LIN {X 0,Y 436.626,Z 302.642,A -85,B 0,C 180,E1 -16932.037,E2 -16932.037} C_VEL
LIN {X 0,Y 436.568,Z 302.656,A -85,B 0,C 180,E1 -16935.718,E2 -16935.718} C_VEL
LIN {X 0,Y 436.534,Z 302.659,A -85,B 0,C 180,E1 -16938.803,E2 -16938.803} C_VEL
LIN {X 0,Y 436.465,Z 302.663,A -85,B 0,C 180,E1 -16941.661,E2 -16941.661} C_VEL
LIN {X 0,Y 436.431,Z 302.68,A -85,B 0,C 180,E1 -16944.663,E2 -16944.663} C_VEL
LIN {X 0,Y 436.477,Z 302.669,A -85,B 0,C 180,E1 -16947.735,E2 -16947.735} C_VEL
LIN {X 0,Y 436.459,Z 302.67,A -85,B 0,C 180,E1 -16950.9,E2 -16950.9} C_VEL
LIN {X 0,Y 436.467,Z 302.658,A -85,B 0,C 180,E1 -16954.172,E2 -16954.172} C_VEL
LIN {X 0,Y 436.511,Z 302.66,A -85,B 0,C 180,E1 -16957.573,E2 -16957.573} C_VEL
LIN {X 0,Y 436.464,Z 302.674,A -85,B 0,C 180,E1 -16961.043,E2 -16961.043} C_VEL
LIN {X 0,Y 436.453,Z 302.675,A -85,B 0,C 180,E1 -16963.769,E2 -16963.769} C_VEL
LIN {X 0,Y 436.456,Z 302.678,A -85,B 0,C 180,E1 -16966.367,E2 -16966.367} C_VEL
LIN {X 0,Y 436.474,Z 302.672,A -85,B 0,C 180,E1 -16968.96,E2 -16968.96} C_VEL
LIN {X 0,Y 436.511,Z 302.67,A -85,B 0,C 180,E1 -16972.431,E2 -16972.431} C_VEL
LIN {X 0,Y 436.473,Z 302.675,A -85,B 0,C 180,E1 -16975.832,E2 -16975.832} C_VEL
LIN {X 0,Y 436.527,Z 302.878,A -85,B 0,C 180,E1 -16976.701,E2 -16976.701} C_VEL
LIN {X 0,Y 439.17,Z 313.579,A -85,B 0,C 180,E1 -16979.048,E2 -16979.048} C_VEL
LIN {X 0,Y 442.005,Z 325.849,A -85,B 0,C 180,E1 -16981.617,E2 -16981.617} C_VEL
LIN {X 0,Y 443.65,Z 334.082,A -85,B 0,C 180,E1 -16983.262,E2 -16983.262} C_VEL
LIN {X 0,Y 443.2,Z 339.732,A -85,B 0,C 180,E1 -16984.269,E2 -16984.269} C_VEL
LIN {X 0,Y 441.528,Z 353.315,A -85,B 0,C 180,E1 -16986.606,E2 -16986.606} C_VEL
LIN {X 0,Y 446.637,Z 380.69,A -85,B 0,C 180,E1 -16987.421,E2 -16987.421} C_VEL
LIN {X 0,Y 449.876,Z 402.607,A -85,B 0,C 180,E1 -16988.005,E2 -16988.005} C_VEL
LIN {X 0,Y 448.042,Z 491.581,A -85,B 0,C 180,E1 -16989.468,E2 -16989.468} C_VEL
LIN {X 0,Y 447.149,Z 506.11,A -85,B 0,C 180,E1 -16989.874,E2 -16989.874} C_VEL
LIN {X 0,Y 445.901,Z 520.039,A -85,B 0,C 180,E1 -16990.443,E2 -16990.443} C_VEL
LIN {X 0,Y 444.716,Z 532.023,A -85,B 0,C 180,E1 -16991.1,E2 -16991.1} C_VEL
LIN {X 0,Y 443.3,Z 544.152,A -85,B 0,C 180,E1 -16991.938,E2 -16991.938} C_VEL
LIN {X 0,Y 441.733,Z 555.894,A -85,B 0,C 180,E1 -16992.944,E2 -16992.944} C_VEL
LIN {X 0,Y 440.163,Z 566.666,A -85,B 0,C 180,E1 -16994.07,E2 -16994.07} C_VEL
LIN {X 0,Y 438.61,Z 577.353,A -85,B 0,C 180,E1 -16995.435,E2 -16995.435} C_VEL
LIN {X 0,Y 437.396,Z 586.21,A -85,B 0,C 180,E1 -16996.811,E2 -16996.811} C_VEL
LIN {X 0,Y 436.36,Z 594.06,A -85,B 0,C 180,E1 -16998.286,E2 -16998.286} C_VEL
LIN {X 0,Y 435.482,Z 600.731,A -85,B 0,C 180,E1 -16999.812,E2 -16999.812} C_VEL
LIN {X 0,Y 434.977,Z 605.724,A -85,B 0,C 180,E1 -17001.203,E2 -17001.203} C_VEL
LIN {X 0,Y 434.568,Z 610.914,A -85,B 0,C 180,E1 -17003.059,E2 -17003.059} C_VEL
LIN {X 0,Y 434.535,Z 612.949,A -85,B 0,C 180,E1 -17003.988,E2 -17003.988} C_VEL
LIN {X 0,Y 434.452,Z 617.176,A -85,B 0,C 180,E1 -17005.379,E2 -17005.379} C_VEL
LIN {X 0,Y 434.447,Z 621.405,A -85,B 0,C 180,E1 -17007.23,E2 -17007.23} C_VEL
LIN {X 0,Y 434.461,Z 624.028,A -85,B 0,C 180,E1 -17009.078,E2 -17009.078} C_VEL
LIN {X 0,Y 434.421,Z 625.147,A -85,B 0,C 180,E1 -17010.926,E2 -17010.926} C_VEL
LIN {X 0,Y 434.377,Z 624.813,A -85,B 0,C 180,E1 -17012.775,E2 -17012.775} C_VEL
LIN {X 0,Y 434.433,Z 623.036,A -85,B 0,C 180,E1 -17014.626,E2 -17014.626} C_VEL
LIN {X 0,Y 434.655,Z 619.805,A -85,B 0,C 180,E1 -17016.479,E2 -17016.479} C_VEL
LIN {X 0,Y 435.059,Z 615.026,A -85,B 0,C 180,E1 -17018.334,E2 -17018.334} C_VEL
LIN {X 0,Y 435.962,Z 608.502,A -85,B 0,C 180,E1 -17020.182,E2 -17020.182} C_VEL
LIN {X 0,Y 436.761,Z 602.482,A -85,B 0,C 180,E1 -17021.552,E2 -17021.552} C_VEL
LIN {X 0,Y 437.804,Z 595.077,A -85,B 0,C 180,E1 -17022.945,E2 -17022.945} C_VEL
LIN {X 0,Y 439.067,Z 586.283,A -85,B 0,C 180,E1 -17024.318,E2 -17024.318} C_VEL
LIN {X 0,Y 440.576,Z 575.698,A -85,B 0,C 180,E1 -17025.683,E2 -17025.683} C_VEL
LIN {X 0,Y 442.174,Z 563.937,A -85,B 0,C 180,E1 -17026.924,E2 -17026.924} C_VEL
LIN {X 0,Y 443.635,Z 552.309,A -85,B 0,C 180,E1 -17027.934,E2 -17027.934} C_VEL
LIN {X 0,Y 445.171,Z 539.699,A -85,B 0,C 180,E1 -17028.819,E2 -17028.819} C_VEL
LIN {X 0,Y 446.569,Z 525.705,A -85,B 0,C 180,E1 -17029.592,E2 -17029.592} C_VEL
LIN {X 0,Y 447.915,Z 510.572,A -85,B 0,C 180,E1 -17030.205,E2 -17030.205} C_VEL
LIN {X 0,Y 448.886,Z 495.971,A -85,B 0,C 180,E1 -17030.615,E2 -17030.615} C_VEL
LIN {X 0,Y 453.117,Z 405.026,A -85,B 0,C 180,E1 -17032.685,E2 -17032.685} C_VEL
LIN {X 0,Y 452.117,Z 390.827,A -85,B 0,C 180,E1 -17033.164,E2 -17033.164} C_VEL
LIN {X 0,Y 449.353,Z 368.94,A -85,B 0,C 180,E1 -17034.04,E2 -17034.04} C_VEL
LIN {X 0,Y 446.685,Z 353.618,A -85,B 0,C 180,E1 -17034.77,E2 -17034.77} C_VEL
LIN {X 0,Y 445.256,Z 335.993,A -85,B 0,C 180,E1 -17036.136,E2 -17036.136} C_VEL
LIN {X 0,Y 444.74,Z 331.395,A -85,B 0,C 180,E1 -17036.538,E2 -17036.538} C_VEL
LIN {X 0,Y 441.955,Z 321.414,A -85,B 0,C 180,E1 -17037.67,E2 -17037.67} C_VEL
LIN {X 0,Y 439.505,Z 312.443,A -85,B 0,C 180,E1 -17038.772,E2 -17038.772} C_VEL
LIN {X 0,Y 436.449,Z 302.672,A -85,B 0,C 180,E1 -17040.194,E2 -17040.194} C_VEL
LIN {X 0,Y 436.409,Z 302.682,A -85,B 0,C 180,E1 -17043.425,E2 -17043.425} C_VEL
LIN {X 0,Y 436.427,Z 302.679,A -85,B 0,C 180,E1 -17046.633,E2 -17046.633} C_VEL
LIN {X 0,Y 436.422,Z 302.681,A -85,B 0,C 180,E1 -17049.942,E2 -17049.942} C_VEL
LIN {X 0,Y 436.438,Z 302.675,A -85,B 0,C 180,E1 -17052.417,E2 -17052.417} C_VEL
LIN {X 0,Y 436.447,Z 302.675,A -85,B 0,C 180,E1 -17055.078,E2 -17055.078} C_VEL
LIN {X 0,Y 436.444,Z 302.678,A -85,B 0,C 180,E1 -17057.619,E2 -17057.619} C_VEL
LIN {X 0,Y 436.427,Z 302.679,A -85,B 0,C 180,E1 -17061.249,E2 -17061.249} C_VEL
LIN {X 0,Y 436.476,Z 302.673,A -85,B 0,C 180,E1 -17064.71,E2 -17064.71} C_VEL
LIN {X 0,Y 436.458,Z 302.676,A -85,B 0,C 180,E1 -17068.022,E2 -17068.022} C_VEL
LIN {X 0,Y 436.479,Z 302.672,A -85,B 0,C 180,E1 -17071.221,E2 -17071.221} C_VEL
LIN {X 0,Y 436.496,Z 302.674,A -85,B 0,C 180,E1 -17074.325,E2 -17074.325} C_VEL
LIN {X 0,Y 436.472,Z 302.681,A -85,B 0,C 180,E1 -17077.347,E2 -17077.347} C_VEL
LIN {X 0,Y 436.481,Z 302.683,A -85,B 0,C 180,E1 -17078.216,E2 -17078.216} C_VEL
LIN {X 0,Y 440.844,Z 314.669,A -85,B 0,C 180,E1 -17081.122,E2 -17081.122} C_VEL
LIN {X 0,Y 444.22,Z 325.795,A -85,B 0,C 180,E1 -17083.511,E2 -17083.511} C_VEL
LIN {X 0,Y 446.243,Z 334.289,A -85,B 0,C 180,E1 -17085.222,E2 -17085.222} C_VEL
LIN {X 0,Y 447.426,Z 340.622,A -85,B 0,C 180,E1 -17086.419,E2 -17086.419} C_VEL
LIN {X 0,Y 447.212,Z 346.49,A -85,B 0,C 180,E1 -17087.349,E2 -17087.349} C_VEL
LIN {X 0,Y 451.527,Z 364.842,A -85,B 0,C 180,E1 -17088.295,E2 -17088.295} C_VEL
LIN {X 0,Y 454.498,Z 381.263,A -85,B 0,C 180,E1 -17089.022,E2 -17089.022} C_VEL
LIN {X 0,Y 449.365,Z 487.032,A -85,B 0,C 180,E1 -17091.428,E2 -17091.428} C_VEL
LIN {X 0,Y 448.385,Z 501.083,A -85,B 0,C 180,E1 -17091.918,E2 -17091.918} C_VEL
LIN {X 0,Y 447.199,Z 514.804,A -85,B 0,C 180,E1 -17092.575,E2 -17092.575} C_VEL
LIN {X 0,Y 445.819,Z 527.476,A -85,B 0,C 180,E1 -17093.346,E2 -17093.346} C_VEL
LIN {X 0,Y 444.246,Z 540.525,A -85,B 0,C 180,E1 -17094.345,E2 -17094.345} C_VEL
LIN {X 0,Y 442.649,Z 552.76,A -85,B 0,C 180,E1 -17095.508,E2 -17095.508} C_VEL
LIN {X 0,Y 441.127,Z 563.905,A -85,B 0,C 180,E1 -17096.814,E2 -17096.814} C_VEL
LIN {X 0,Y 439.628,Z 573.517,A -85,B 0,C 180,E1 -17098.174,E2 -17098.174} C_VEL
LIN {X 0,Y 438.204,Z 581.565,A -85,B 0,C 180,E1 -17099.542,E2 -17099.542} C_VEL
LIN {X 0,Y 437.03,Z 589.247,A -85,B 0,C 180,E1 -17101.148,E2 -17101.148} C_VEL
LIN {X 0,Y 436.08,Z 595.41,A -85,B 0,C 180,E1 -17102.762,E2 -17102.762} C_VEL
LIN {X 0,Y 435.53,Z 600.07,A -85,B 0,C 180,E1 -17104.332,E2 -17104.332} C_VEL
LIN {X 0,Y 435.12,Z 602.903,A -85,B 0,C 180,E1 -17105.543,E2 -17105.543} C_VEL
LIN {X 0,Y 434.602,Z 605.961,A -85,B 0,C 180,E1 -17107.408,E2 -17107.408} C_VEL
LIN {X 0,Y 434.369,Z 607.556,A -85,B 0,C 180,E1 -17109.28,E2 -17109.28} C_VEL
LIN {X 0,Y 434.327,Z 607.829,A -85,B 0,C 180,E1 -17110.335,E2 -17110.335} C_VEL
LIN {X 0,Y 434.162,Z 607.229,A -85,B 0,C 180,E1 -17112.107,E2 -17112.107} C_VEL
LIN {X 0,Y 434.186,Z 606.372,A -85,B 0,C 180,E1 -17113.053,E2 -17113.053} C_VEL
LIN {X 0,Y 434.297,Z 604.126,A -85,B 0,C 180,E1 -17114.598,E2 -17114.598} C_VEL
LIN {X 0,Y 434.384,Z 600.223,A -85,B 0,C 180,E1 -17116.391,E2 -17116.391} C_VEL
LIN {X 0,Y 434.608,Z 595.302,A -85,B 0,C 180,E1 -17118.028,E2 -17118.028} C_VEL
LIN {X 0,Y 434.948,Z 588.493,A -85,B 0,C 180,E1 -17119.766,E2 -17119.766} C_VEL
LIN {X 0,Y 435.348,Z 580.859,A -85,B 0,C 180,E1 -17121.322,E2 -17121.322} C_VEL
LIN {X 0,Y 435.846,Z 572.726,A -85,B 0,C 180,E1 -17122.687,E2 -17122.687} C_VEL
LIN {X 0,Y 436.535,Z 562.361,A -85,B 0,C 180,E1 -17124.128,E2 -17124.128} C_VEL
LIN {X 0,Y 437.273,Z 551.493,A -85,B 0,C 180,E1 -17125.372,E2 -17125.372} C_VEL
LIN {X 0,Y 438.069,Z 539.353,A -85,B 0,C 180,E1 -17126.509,E2 -17126.509} C_VEL
LIN {X 0,Y 438.8,Z 527.117,A -85,B 0,C 180,E1 -17127.447,E2 -17127.447} C_VEL
LIN {X 0,Y 439.547,Z 513.158,A -85,B 0,C 180,E1 -17128.3,E2 -17128.3} C_VEL
LIN {X 0,Y 440.253,Z 499.336,A -85,B 0,C 180,E1 -17128.946,E2 -17128.946} C_VEL
LIN {X 0,Y 440.866,Z 484.516,A -85,B 0,C 180,E1 -17129.439,E2 -17129.439} C_VEL
LIN {X 0,Y 443.335,Z 374.69,A -85,B 0,C 180,E1 -17131.717,E2 -17131.717} C_VEL
LIN {X 0,Y 439.387,Z 344.217,A -85,B 0,C 180,E1 -17132.505,E2 -17132.505} C_VEL
LIN {X 0,Y 440.404,Z 324.501,A -85,B 0,C 180,E1 -17135.487,E2 -17135.487} C_VEL
LIN {X 0,Y 440.116,Z 320.765,A -85,B 0,C 180,E1 -17136.076,E2 -17136.076} C_VEL
LIN {X 0,Y 436.475,Z 302.673,A -85,B 0,C 180,E1 -17139.041,E2 -17139.041} C_VEL
LIN {X 0,Y 436.451,Z 302.68,A -85,B 0,C 180,E1 -17142.416,E2 -17142.416} C_VEL
LIN {X 0,Y 436.444,Z 302.673,A -85,B 0,C 180,E1 -17145.075,E2 -17145.075} C_VEL
LIN {X 0,Y 436.443,Z 302.674,A -85,B 0,C 180,E1 -17147.617,E2 -17147.617} C_VEL
LIN {X 0,Y 436.414,Z 302.677,A -85,B 0,C 180,E1 -17151.246,E2 -17151.246} C_VEL
LIN {X 0,Y 436.418,Z 302.678,A -85,B 0,C 180,E1 -17154.702,E2 -17154.702} C_VEL
LIN {X 0,Y 436.427,Z 302.681,A -85,B 0,C 180,E1 -17158.017,E2 -17158.017} C_VEL
LIN {X 0,Y 436.462,Z 302.67,A -85,B 0,C 180,E1 -17161.218,E2 -17161.218} C_VEL
LIN {X 0,Y 436.47,Z 302.674,A -85,B 0,C 180,E1 -17164.321,E2 -17164.321} C_VEL
LIN {X 0,Y 436.468,Z 302.671,A -85,B 0,C 180,E1 -17167.345,E2 -17167.345} C_VEL
LIN {X 0,Y 436.525,Z 302.666,A -85,B 0,C 180,E1 -17170.306,E2 -17170.306} C_VEL
LIN {X 0,Y 436.518,Z 302.664,A -85,B 0,C 180,E1 -17173.21,E2 -17173.21} C_VEL
LIN {X 0,Y 436.586,Z 302.656,A -85,B 0,C 180,E1 -17175.124,E2 -17175.124} C_VEL
LIN {X 0,Y 436.637,Z 302.654,A -85,B 0,C 180,E1 -17178.111,E2 -17178.111} C_VEL
LIN {X 0,Y 436.606,Z 302.66,A -85,B 0,C 180,E1 -17180.125,E2 -17180.125} C_VEL
LIN {X 0,Y 437.575,Z 307.511,A -85,B 0,C 180,E1 -17181.195,E2 -17181.195} C_VEL
LIN {X 0,Y 442.962,Z 324.717,A -85,B 0,C 180,E1 -17181.703,E2 -17181.703} C_VEL
LIN {X 0,Y 444.742,Z 334.457,A -85,B 0,C 180,E1 -17181.935,E2 -17181.935} C_VEL
LIN {X 0,Y 442.794,Z 443.192,A -85,B 0,C 180,E1 -17183.697,E2 -17183.697} C_VEL
LIN {X 0,Y 442.407,Z 457.507,A -85,B 0,C 180,E1 -17184.12,E2 -17184.12} C_VEL
LIN {X 0,Y 441.822,Z 471.29,A -85,B 0,C 180,E1 -17184.711,E2 -17184.711} C_VEL
LIN {X 0,Y 441.087,Z 484.15,A -85,B 0,C 180,E1 -17185.444,E2 -17185.444} C_VEL
LIN {X 0,Y 440.265,Z 496.628,A -85,B 0,C 180,E1 -17186.349,E2 -17186.349} C_VEL
LIN {X 0,Y 439.176,Z 508.084,A -85,B 0,C 180,E1 -17187.37,E2 -17187.37} C_VEL
LIN {X 0,Y 438.531,Z 517.551,A -85,B 0,C 180,E1 -17188.396,E2 -17188.396} C_VEL
LIN {X 0,Y 437.726,Z 526.51,A -85,B 0,C 180,E1 -17189.539,E2 -17189.539} C_VEL
LIN {X 0,Y 436.853,Z 535.526,A -85,B 0,C 180,E1 -17190.916,E2 -17190.916} C_VEL
LIN {X 0,Y 436.202,Z 543.032,A -85,B 0,C 180,E1 -17192.298,E2 -17192.298} C_VEL
LIN {X 0,Y 435.769,Z 549.294,A -85,B 0,C 180,E1 -17193.684,E2 -17193.684} C_VEL
LIN {X 0,Y 435.424,Z 554.44,A -85,B 0,C 180,E1 -17195.074,E2 -17195.074} C_VEL
LIN {X 0,Y 434.989,Z 559.886,A -85,B 0,C 180,E1 -17196.934,E2 -17196.934} C_VEL
LIN {X 0,Y 434.719,Z 562.912,A -85,B 0,C 180,E1 -17198.336,E2 -17198.336} C_VEL
LIN {X 0,Y 434.676,Z 565.728,A -85,B 0,C 180,E1 -17200.207,E2 -17200.207} C_VEL
LIN {X 0,Y 434.605,Z 567.192,A -85,B 0,C 180,E1 -17202.092,E2 -17202.092} C_VEL
LIN {X 0,Y 434.789,Z 567.295,A -85,B 0,C 180,E1 -17203.981,E2 -17203.981} C_VEL
LIN {X 0,Y 434.933,Z 566.595,A -85,B 0,C 180,E1 -17205.208,E2 -17205.208} C_VEL
LIN {X 0,Y 434.374,Z 565.963,A -85,B 0,C 180,E1 -17205.977,E2 -17205.977} C_VEL
LIN {X 0,Y 431.785,Z 564.572,A -85,B 0,C 180,E1 -17207.231,E2 -17207.231} C_VEL
LIN {X 0,Y 429.673,Z 563.1,A -85,B 0,C 180,E1 -17208.232,E2 -17208.232} C_VEL
LIN {X 0,Y 428.912,Z 561.668,A -85,B 0,C 180,E1 -17208.991,E2 -17208.991} C_VEL
LIN {X 0,Y 428.929,Z 561.104,A -85,B 0,C 180,E1 -17209.244,E2 -17209.244} C_VEL
LIN {X 0,Y 429.778,Z 556.392,A -85,B 0,C 180,E1 -17211.008,E2 -17211.008} C_VEL
LIN {X 0,Y 430.608,Z 551.365,A -85,B 0,C 180,E1 -17212.471,E2 -17212.471} C_VEL
LIN {X 0,Y 431.869,Z 544.086,A -85,B 0,C 180,E1 -17214.172,E2 -17214.172} C_VEL
LIN {X 0,Y 433.184,Z 536.526,A -85,B 0,C 180,E1 -17215.6,E2 -17215.6} C_VEL
LIN {X 0,Y 434.655,Z 527.055,A -85,B 0,C 180,E1 -17217.078,E2 -17217.078} C_VEL
LIN {X 0,Y 436.234,Z 516.669,A -85,B 0,C 180,E1 -17218.4,E2 -17218.4} C_VEL
LIN {X 0,Y 437.768,Z 505.104,A -85,B 0,C 180,E1 -17219.601,E2 -17219.601} C_VEL
LIN {X 0,Y 439.125,Z 493.279,A -85,B 0,C 180,E1 -17220.598,E2 -17220.598} C_VEL
LIN {X 0,Y 440.386,Z 480.518,A -85,B 0,C 180,E1 -17221.456,E2 -17221.456} C_VEL
LIN {X 0,Y 441.357,Z 466.602,A -85,B 0,C 180,E1 -17222.181,E2 -17222.181} C_VEL
LIN {X 0,Y 442.137,Z 452.151,A -85,B 0,C 180,E1 -17222.721,E2 -17222.721} C_VEL
LIN {X 0,Y 442.67,Z 437.341,A -85,B 0,C 180,E1 -17223.068,E2 -17223.068} C_VEL
LIN {X 0,Y 444.754,Z 341.078,A -85,B 0,C 180,E1 -17224.648,E2 -17224.648} C_VEL
LIN {X 0,Y 437.111,Z 323.008,A -85,B 0,C 180,E1 -17225.488,E2 -17225.488} C_VEL
LIN {X 0,Y 430.623,Z 308.973,A -85,B 0,C 180,E1 -17226.215,E2 -17226.215} C_VEL
LIN {X 0,Y 429.394,Z 303.558,A -85,B 0,C 180,E1 -17227.71,E2 -17227.71} C_VEL
LIN {X 0,Y 429.355,Z 303.557,A -85,B 0,C 180,E1 -17230.731,E2 -17230.731} C_VEL
LIN {X 0,Y 429.384,Z 303.547,A -85,B 0,C 180,E1 -17234.13,E2 -17234.13} C_VEL
LIN {X 0,Y 429.363,Z 303.56,A -85,B 0,C 180,E1 -17237.228,E2 -17237.228} C_VEL
LIN {X 0,Y 429.369,Z 303.556,A -85,B 0,C 180,E1 -17240.489,E2 -17240.489} C_VEL
LIN {X 0,Y 429.396,Z 303.529,A -85,B 0,C 180,E1 -17244.038,E2 -17244.038} C_VEL
LIN {X 0,Y 429.374,Z 303.559,A -85,B 0,C 180,E1 -17247.43,E2 -17247.43} C_VEL
LIN {X 0,Y 429.405,Z 303.553,A -85,B 0,C 180,E1 -17250.702,E2 -17250.702} C_VEL
LIN {X 0,Y 429.433,Z 303.55,A -85,B 0,C 180,E1 -17253.871,E2 -17253.871} C_VEL
LIN {X 0,Y 429.426,Z 303.54,A -85,B 0,C 180,E1 -17256.954,E2 -17256.954} C_VEL
LIN {X 0,Y 429.444,Z 303.543,A -85,B 0,C 180,E1 -17259.97,E2 -17259.97} C_VEL
LIN {X 0,Y 429.414,Z 303.55,A -85,B 0,C 180,E1 -17262.926,E2 -17262.926} C_VEL
LIN {X 0,Y 429.503,Z 303.529,A -85,B 0,C 180,E1 -17265.84,E2 -17265.84} C_VEL
LIN {X 0,Y 429.583,Z 303.531,A -85,B 0,C 180,E1 -17268.717,E2 -17268.717} C_VEL
LIN {X 0,Y 429.622,Z 303.521,A -85,B 0,C 180,E1 -17272.506,E2 -17272.506} C_VEL
LIN {X 0,Y 429.735,Z 303.503,A -85,B 0,C 180,E1 -17275.325,E2 -17275.325} C_VEL
LIN {X 0,Y 429.646,Z 303.527,A -85,B 0,C 180,E1 -17279.066,E2 -17279.066} C_VEL
LIN {X 0,Y 429.638,Z 303.515,A -85,B 0,C 180,E1 -17280.934,E2 -17280.934} C_VEL
LIN {X 0,Y 429.765,Z 303.509,A -85,B 0,C 180,E1 -17284.674,E2 -17284.674} C_VEL
LIN {X 0,Y 429.624,Z 303.511,A -85,B 0,C 180,E1 -17287.494,E2 -17287.494} C_VEL
LIN {X 0,Y 429.63,Z 303.516,A -85,B 0,C 180,E1 -17291.282,E2 -17291.282} C_VEL
LIN {X 0,Y 429.527,Z 303.536,A -85,B 0,C 180,E1 -17295.125,E2 -17295.125} C_VEL
LIN {X 0,Y 429.483,Z 303.539,A -85,B 0,C 180,E1 -17298.939,E2 -17298.939} C_VEL
LIN {X 0,Y 429.423,Z 303.54,A -85,B 0,C 180,E1 -17302.034,E2 -17302.034} C_VEL
LIN {X 0,Y 429.39,Z 303.552,A -85,B 0,C 180,E1 -17305.095,E2 -17305.095} C_VEL
LIN {X 0,Y 429.434,Z 303.55,A -85,B 0,C 180,E1 -17308.269,E2 -17308.269} C_VEL
LIN {X 0,Y 429.428,Z 303.547,A -85,B 0,C 180,E1 -17311.464,E2 -17311.464} C_VEL
LIN {X 0,Y 429.426,Z 303.525,A -85,B 0,C 180,E1 -17314.812,E2 -17314.812} C_VEL
LIN {X 0,Y 429.463,Z 303.53,A -85,B 0,C 180,E1 -17317.118,E2 -17317.118} C_VEL
LIN {X 0,Y 429.435,Z 303.548,A -85,B 0,C 180,E1 -17319.954,E2 -17319.954} C_VEL
LIN {X 0,Y 429.414,Z 303.55,A -85,B 0,C 180,E1 -17323.243,E2 -17323.243} C_VEL
LIN {X 0,Y 429.416,Z 303.551,A -85,B 0,C 180,E1 -17326.762,E2 -17326.762} C_VEL
LIN {X 0,Y 429.432,Z 303.553,A -85,B 0,C 180,E1 -17330.051,E2 -17330.051} C_VEL
LIN {X 0,Y 429.468,Z 303.541,A -85,B 0,C 180,E1 -17333.051,E2 -17333.051} C_VEL
LIN {X 0,Y 429.458,Z 303.663,A -85,B 0,C 180,E1 -17336.23,E2 -17336.23} C_VEL
LIN {X 0,Y 431.987,Z 313.599,A -85,B 0,C 180,E1 -17338.475,E2 -17338.475} C_VEL
LIN {X 0,Y 435.095,Z 327.249,A -85,B 0,C 180,E1 -17341.387,E2 -17341.387} C_VEL
LIN {X 0,Y 436.884,Z 336.795,A -85,B 0,C 180,E1 -17343.329,E2 -17343.329} C_VEL
LIN {X 0,Y 434.91,Z 351.918,A -85,B 0,C 180,E1 -17346.007,E2 -17346.007} C_VEL
LIN {X 0,Y 434.807,Z 352.7,A -85,B 0,C 180,E1 -17346.143,E2 -17346.143} C_VEL
LIN {X 0,Y 439.93,Z 379.664,A -85,B 0,C 180,E1 -17346.975,E2 -17346.975} C_VEL
LIN {X 0,Y 443.54,Z 403.892,A -85,B 0,C 180,E1 -17347.637,E2 -17347.637} C_VEL
LIN {X 0,Y 441.56,Z 491.392,A -85,B 0,C 180,E1 -17349.092,E2 -17349.092} C_VEL
LIN {X 0,Y 440.653,Z 505.836,A -85,B 0,C 180,E1 -17349.503,E2 -17349.503} C_VEL
LIN {X 0,Y 439.387,Z 519.478,A -85,B 0,C 180,E1 -17350.068,E2 -17350.068} C_VEL
LIN {X 0,Y 437.98,Z 533.01,A -85,B 0,C 180,E1 -17350.829,E2 -17350.829} C_VEL
LIN {X 0,Y 436.394,Z 545.908,A -85,B 0,C 180,E1 -17351.763,E2 -17351.763} C_VEL
LIN {X 0,Y 434.66,Z 558.428,A -85,B 0,C 180,E1 -17352.899,E2 -17352.899} C_VEL
LIN {X 0,Y 433.008,Z 568.701,A -85,B 0,C 180,E1 -17354.041,E2 -17354.041} C_VEL
LIN {X 0,Y 431.489,Z 578.968,A -85,B 0,C 180,E1 -17355.43,E2 -17355.43} C_VEL
LIN {X 0,Y 430.283,Z 587.492,A -85,B 0,C 180,E1 -17356.829,E2 -17356.829} C_VEL
LIN {X 0,Y 429.109,Z 595.849,A -85,B 0,C 180,E1 -17358.507,E2 -17358.507} C_VEL
LIN {X 0,Y 428.267,Z 602.319,A -85,B 0,C 180,E1 -17360.114,E2 -17360.114} C_VEL
LIN {X 0,Y 427.63,Z 608.251,A -85,B 0,C 180,E1 -17361.999,E2 -17361.999} C_VEL
LIN {X 0,Y 427.429,Z 613.872,A -85,B 0,C 180,E1 -17364.36,E2 -17364.36} C_VEL
LIN {X 0,Y 427.341,Z 617.927,A -85,B 0,C 180,E1 -17365.772,E2 -17365.772} C_VEL
LIN {X 0,Y 427.369,Z 620.993,A -85,B 0,C 180,E1 -17367.184,E2 -17367.184} C_VEL
LIN {X 0,Y 427.369,Z 623.747,A -85,B 0,C 180,E1 -17369.063,E2 -17369.063} C_VEL
LIN {X 0,Y 427.329,Z 624.97,A -85,B 0,C 180,E1 -17370.941,E2 -17370.941} C_VEL
LIN {X 0,Y 427.275,Z 624.724,A -85,B 0,C 180,E1 -17372.821,E2 -17372.821} C_VEL
LIN {X 0,Y 427.356,Z 623.04,A -85,B 0,C 180,E1 -17374.703,E2 -17374.703} C_VEL
LIN {X 0,Y 427.593,Z 619.894,A -85,B 0,C 180,E1 -17376.587,E2 -17376.587} C_VEL
LIN {X 0,Y 428.021,Z 615.234,A -85,B 0,C 180,E1 -17378.472,E2 -17378.472} C_VEL
LIN {X 0,Y 428.721,Z 610.605,A -85,B 0,C 180,E1 -17379.88,E2 -17379.88} C_VEL
LIN {X 0,Y 429.726,Z 603.921,A -85,B 0,C 180,E1 -17381.52,E2 -17381.52} C_VEL
LIN {X 0,Y 430.69,Z 597.062,A -85,B 0,C 180,E1 -17382.9,E2 -17382.9} C_VEL
LIN {X 0,Y 431.96,Z 588.565,A -85,B 0,C 180,E1 -17384.319,E2 -17384.319} C_VEL
LIN {X 0,Y 433.551,Z 578.519,A -85,B 0,C 180,E1 -17385.703,E2 -17385.703} C_VEL
LIN {X 0,Y 435.098,Z 567.471,A -85,B 0,C 180,E1 -17386.967,E2 -17386.967} C_VEL
LIN {X 0,Y 436.801,Z 555.205,A -85,B 0,C 180,E1 -17388.103,E2 -17388.103} C_VEL
LIN {X 0,Y 438.591,Z 541.584,A -85,B 0,C 180,E1 -17389.113,E2 -17389.113} C_VEL
LIN {X 0,Y 440.16,Z 527.083,A -85,B 0,C 180,E1 -17389.962,E2 -17389.962} C_VEL
LIN {X 0,Y 441.569,Z 512.368,A -85,B 0,C 180,E1 -17390.59,E2 -17390.59} C_VEL
LIN {X 0,Y 442.673,Z 497.253,A -85,B 0,C 180,E1 -17391.04,E2 -17391.04} C_VEL
LIN {X 0,Y 447.215,Z 404.968,A -85,B 0,C 180,E1 -17393.194,E2 -17393.194} C_VEL
LIN {X 0,Y 446.004,Z 389.679,A -85,B 0,C 180,E1 -17393.745,E2 -17393.745} C_VEL
LIN {X 0,Y 443.582,Z 370.493,A -85,B 0,C 180,E1 -17394.546,E2 -17394.546} C_VEL
LIN {X 0,Y 440.73,Z 353.693,A -85,B 0,C 180,E1 -17395.362,E2 -17395.362} C_VEL
LIN {X 0,Y 439.433,Z 336.148,A -85,B 0,C 180,E1 -17396.795,E2 -17396.795} C_VEL
LIN {X 0,Y 437.214,Z 326.969,A -85,B 0,C 180,E1 -17397.815,E2 -17397.815} C_VEL
LIN {X 0,Y 434.45,Z 316.696,A -85,B 0,C 180,E1 -17399.107,E2 -17399.107} C_VEL
LIN {X 0,Y 431.918,Z 308.732,A -85,B 0,C 180,E1 -17400.281,E2 -17400.281} C_VEL
LIN {X 0,Y 429.869,Z 305.411,A -85,B 0,C 180,E1 -17400.975,E2 -17400.975} C_VEL
LIN {X 0,Y 429.39,Z 303.559,A -85,B 0,C 180,E1 -17401.296,E2 -17401.296} C_VEL
LIN {X 0,Y 429.358,Z 303.562,A -85,B 0,C 180,E1 -17404.821,E2 -17404.821} C_VEL
LIN {X 0,Y 429.395,Z 303.556,A -85,B 0,C 180,E1 -17407.127,E2 -17407.127} C_VEL
LIN {X 0,Y 429.374,Z 303.557,A -85,B 0,C 180,E1 -17410.734,E2 -17410.734} C_VEL
LIN {X 0,Y 429.404,Z 303.552,A -85,B 0,C 180,E1 -17414.133,E2 -17414.133} C_VEL
LIN {X 0,Y 429.377,Z 303.557,A -85,B 0,C 180,E1 -17417.232,E2 -17417.232} C_VEL
LIN {X 0,Y 429.377,Z 303.558,A -85,B 0,C 180,E1 -17420.49,E2 -17420.49} C_VEL
LIN {X 0,Y 429.418,Z 303.554,A -85,B 0,C 180,E1 -17424.04,E2 -17424.04} C_VEL
LIN {X 0,Y 429.416,Z 303.552,A -85,B 0,C 180,E1 -17426.317,E2 -17426.317} C_VEL
LIN {X 0,Y 429.422,Z 303.553,A -85,B 0,C 180,E1 -17429.828,E2 -17429.828} C_VEL
LIN {X 0,Y 429.451,Z 303.549,A -85,B 0,C 180,E1 -17432.826,E2 -17432.826} C_VEL
LIN {X 0,Y 429.461,Z 303.553,A -85,B 0,C 180,E1 -17435.976,E2 -17435.976} C_VEL
LIN {X 0,Y 429.445,Z 303.664,A -85,B 0,C 180,E1 -17437.241,E2 -17437.241} C_VEL
LIN {X 0,Y 432.626,Z 311.957,A -85,B 0,C 180,E1 -17439.419,E2 -17439.419} C_VEL
LIN {X 0,Y 435.921,Z 321.432,A -85,B 0,C 180,E1 -17441.672,E2 -17441.672} C_VEL
LIN {X 0,Y 439.234,Z 333.556,A -85,B 0,C 180,E1 -17444.27,E2 -17444.27} C_VEL
LIN {X 0,Y 441.114,Z 343.482,A -85,B 0,C 180,E1 -17446.221,E2 -17446.221} C_VEL
LIN {X 0,Y 441.051,Z 346.59,A -85,B 0,C 180,E1 -17446.721,E2 -17446.721} C_VEL
LIN {X 0,Y 445.166,Z 363.673,A -85,B 0,C 180,E1 -17447.66,E2 -17447.66} C_VEL
LIN {X 0,Y 448.574,Z 382.224,A -85,B 0,C 180,E1 -17448.523,E2 -17448.523} C_VEL
LIN {X 0,Y 443.749,Z 477.266,A -85,B 0,C 180,E1 -17450.718,E2 -17450.718} C_VEL
LIN {X 0,Y 442.824,Z 492.968,A -85,B 0,C 180,E1 -17451.157,E2 -17451.157} C_VEL
LIN {X 0,Y 441.817,Z 506.013,A -85,B 0,C 180,E1 -17451.682,E2 -17451.682} C_VEL
LIN {X 0,Y 440.558,Z 518.746,A -85,B 0,C 180,E1 -17452.348,E2 -17452.348} C_VEL
LIN {X 0,Y 438.964,Z 532.13,A -85,B 0,C 180,E1 -17453.242,E2 -17453.242} C_VEL
LIN {X 0,Y 437.213,Z 545.475,A -85,B 0,C 180,E1 -17454.369,E2 -17454.369} C_VEL
LIN {X 0,Y 435.599,Z 556.857,A -85,B 0,C 180,E1 -17455.549,E2 -17455.549} C_VEL
LIN {X 0,Y 434.174,Z 566.516,A -85,B 0,C 180,E1 -17456.763,E2 -17456.763} C_VEL
LIN {X 0,Y 432.6,Z 575.74,A -85,B 0,C 180,E1 -17458.144,E2 -17458.144} C_VEL
LIN {X 0,Y 431.176,Z 583.456,A -85,B 0,C 180,E1 -17459.535,E2 -17459.535} C_VEL
LIN {X 0,Y 430.123,Z 589.824,A -85,B 0,C 180,E1 -17460.933,E2 -17460.933} C_VEL
LIN {X 0,Y 429.258,Z 595.093,A -85,B 0,C 180,E1 -17462.338,E2 -17462.338} C_VEL
LIN {X 0,Y 428.621,Z 599.392,A -85,B 0,C 180,E1 -17463.748,E2 -17463.748} C_VEL
LIN {X 0,Y 428.019,Z 603.696,A -85,B 0,C 180,E1 -17465.635,E2 -17465.635} C_VEL
LIN {X 0,Y 427.487,Z 606.516,A -85,B 0,C 180,E1 -17467.532,E2 -17467.532} C_VEL
LIN {X 0,Y 427.274,Z 607.878,A -85,B 0,C 180,E1 -17469.435,E2 -17469.435} C_VEL
LIN {X 0,Y 427.241,Z 608.003,A -85,B 0,C 180,E1 -17470.39,E2 -17470.39} C_VEL
LIN {X 0,Y 427.071,Z 607.118,A -85,B 0,C 180,E1 -17472.311,E2 -17472.311} C_VEL
LIN {X 0,Y 427.171,Z 604.728,A -85,B 0,C 180,E1 -17474.238,E2 -17474.238} C_VEL
LIN {X 0,Y 427.28,Z 600.741,A -85,B 0,C 180,E1 -17476.182,E2 -17476.182} C_VEL
LIN {X 0,Y 427.475,Z 596.567,A -85,B 0,C 180,E1 -17477.646,E2 -17477.646} C_VEL
LIN {X 0,Y 427.742,Z 590.313,A -85,B 0,C 180,E1 -17479.366,E2 -17479.366} C_VEL
LIN {X 0,Y 428.15,Z 583.586,A -85,B 0,C 180,E1 -17480.844,E2 -17480.844} C_VEL
LIN {X 0,Y 428.614,Z 575.375,A -85,B 0,C 180,E1 -17482.331,E2 -17482.331} C_VEL
LIN {X 0,Y 429.291,Z 565.57,A -85,B 0,C 180,E1 -17483.788,E2 -17483.788} C_VEL
LIN {X 0,Y 430.033,Z 554.107,A -85,B 0,C 180,E1 -17485.184,E2 -17485.184} C_VEL
LIN {X 0,Y 430.866,Z 541.786,A -85,B 0,C 180,E1 -17486.411,E2 -17486.411} C_VEL
LIN {X 0,Y 431.62,Z 529.372,A -85,B 0,C 180,E1 -17487.418,E2 -17487.418} C_VEL
LIN {X 0,Y 432.369,Z 515.953,A -85,B 0,C 180,E1 -17488.285,E2 -17488.285} C_VEL
LIN {X 0,Y 433.147,Z 501.099,A -85,B 0,C 180,E1 -17489.021,E2 -17489.021} C_VEL
LIN {X 0,Y 433.828,Z 486.487,A -85,B 0,C 180,E1 -17489.543,E2 -17489.543} C_VEL
LIN {X 0,Y 434.281,Z 464.922,A -85,B 0,C 180,E1 -17490.033,E2 -17490.033} C_VEL
LIN {X 0,Y 436.48,Z 375.925,A -85,B 0,C 180,E1 -17491.894,E2 -17491.894} C_VEL
LIN {X 0,Y 432.438,Z 344.253,A -85,B 0,C 180,E1 -17492.735,E2 -17492.735} C_VEL
LIN {X 0,Y 433.455,Z 324.565,A -85,B 0,C 180,E1 -17495.747,E2 -17495.747} C_VEL
LIN {X 0,Y 431.419,Z 313.227,A -85,B 0,C 180,E1 -17497.592,E2 -17497.592} C_VEL
LIN {X 0,Y 429.424,Z 303.552,A -85,B 0,C 180,E1 -17499.208,E2 -17499.208} C_VEL
LIN {X 0,Y 429.387,Z 303.555,A -85,B 0,C 180,E1 -17502.769,E2 -17502.769} C_VEL
LIN {X 0,Y 429.396,Z 303.552,A -85,B 0,C 180,E1 -17505.868,E2 -17505.868} C_VEL
LIN {X 0,Y 429.374,Z 303.553,A -85,B 0,C 180,E1 -17509.265,E2 -17509.265} C_VEL
LIN {X 0,Y 429.394,Z 303.552,A -85,B 0,C 180,E1 -17512.873,E2 -17512.873} C_VEL
LIN {X 0,Y 429.397,Z 303.556,A -85,B 0,C 180,E1 -17516.314,E2 -17516.314} C_VEL
LIN {X 0,Y 429.411,Z 303.553,A -85,B 0,C 180,E1 -17519.828,E2 -17519.828} C_VEL
LIN {X 0,Y 429.425,Z 303.548,A -85,B 0,C 180,E1 -17522.823,E2 -17522.823} C_VEL
LIN {X 0,Y 429.457,Z 303.55,A -85,B 0,C 180,E1 -17525.974,E2 -17525.974} C_VEL
LIN {X 0,Y 429.461,Z 303.543,A -85,B 0,C 180,E1 -17528.97,E2 -17528.97} C_VEL
LIN {X 0,Y 429.466,Z 303.55,A -85,B 0,C 180,E1 -17531.946,E2 -17531.946} C_VEL
LIN {X 0,Y 429.543,Z 303.533,A -85,B 0,C 180,E1 -17534.874,E2 -17534.874} C_VEL
LIN {X 0,Y 429.611,Z 303.525,A -85,B 0,C 180,E1 -17538.715,E2 -17538.715} C_VEL
LIN {X 0,Y 429.587,Z 303.67,A -85,B 0,C 180,E1 -17539.962,E2 -17539.962} C_VEL
LIN {X 0,Y 430.368,Z 307.586,A -85,B 0,C 180,E1 -17540.885,E2 -17540.885} C_VEL
LIN {X 0,Y 436.359,Z 326.547,A -85,B 0,C 180,E1 -17541.469,E2 -17541.469} C_VEL
LIN {X 0,Y 437.953,Z 334.866,A -85,B 0,C 180,E1 -17541.674,E2 -17541.674} C_VEL
LIN {X 0,Y 435.957,Z 443.291,A -85,B 0,C 180,E1 -17543.453,E2 -17543.453} C_VEL
LIN {X 0,Y 435.556,Z 457.709,A -85,B 0,C 180,E1 -17543.882,E2 -17543.882} C_VEL
LIN {X 0,Y 434.923,Z 472.104,A -85,B 0,C 180,E1 -17544.511,E2 -17544.511} C_VEL
LIN {X 0,Y 434.174,Z 484.873,A -85,B 0,C 180,E1 -17545.255,E2 -17545.255} C_VEL
LIN {X 0,Y 433.305,Z 497.298,A -85,B 0,C 180,E1 -17546.174,E2 -17546.174} C_VEL
LIN {X 0,Y 432.225,Z 508.7,A -85,B 0,C 180,E1 -17547.211,E2 -17547.211} C_VEL
LIN {X 0,Y 431.5,Z 519.095,A -85,B 0,C 180,E1 -17548.37,E2 -17548.37} C_VEL
LIN {X 0,Y 430.444,Z 529.5,A -85,B 0,C 180,E1 -17549.765,E2 -17549.765} C_VEL
LIN {X 0,Y 429.683,Z 538.07,A -85,B 0,C 180,E1 -17551.165,E2 -17551.165} C_VEL
LIN {X 0,Y 428.837,Z 546.319,A -85,B 0,C 180,E1 -17552.806,E2 -17552.806} C_VEL
LIN {X 0,Y 428.544,Z 552.793,A -85,B 0,C 180,E1 -17554.417,E2 -17554.417} C_VEL
LIN {X 0,Y 428.099,Z 558.179,A -85,B 0,C 180,E1 -17556.103,E2 -17556.103} C_VEL
LIN {X 0,Y 427.801,Z 561.693,A -85,B 0,C 180,E1 -17557.524,E2 -17557.524} C_VEL
LIN {X 0,Y 427.599,Z 565.124,A -85,B 0,C 180,E1 -17559.426,E2 -17559.426} C_VEL
LIN {X 0,Y 427.511,Z 567.166,A -85,B 0,C 180,E1 -17561.336,E2 -17561.336} C_VEL
LIN {X 0,Y 427.586,Z 567.834,A -85,B 0,C 180,E1 -17563.256,E2 -17563.256} C_VEL
LIN {X 0,Y 427.859,Z 567.096,A -85,B 0,C 180,E1 -17565.227,E2 -17565.227} C_VEL
LIN {X 0,Y 428.2,Z 565.055,A -85,B 0,C 180,E1 -17567.121,E2 -17567.121} C_VEL
LIN {X 0,Y 428.859,Z 561.514,A -85,B 0,C 180,E1 -17569.063,E2 -17569.063} C_VEL
LIN {X 0,Y 428.929,Z 561.104,A -85,B 0,C 180,E1 -17569.244,E2 -17569.244} C_VEL
LIN {X 0,Y 428.588,Z 559.37,A -85,B 0,C 180,E1 -17569.998,E2 -17569.998} C_VEL
LIN {X 0,Y 426.337,Z 556.295,A -85,B 0,C 180,E1 -17571.226,E2 -17571.226} C_VEL
LIN {X 0,Y 424.185,Z 552.683,A -85,B 0,C 180,E1 -17572.437,E2 -17572.437} C_VEL
LIN {X 0,Y 424.001,Z 550.059,A -85,B 0,C 180,E1 -17573.154,E2 -17573.154} C_VEL
LIN {X 0,Y 425.332,Z 542.951,A -85,B 0,C 180,E1 -17574.761,E2 -17574.761} C_VEL
LIN {X 0,Y 426.772,Z 534.529,A -85,B 0,C 180,E1 -17576.301,E2 -17576.301} C_VEL
LIN {X 0,Y 428.305,Z 525.239,A -85,B 0,C 180,E1 -17577.696,E2 -17577.696} C_VEL
LIN {X 0,Y 429.892,Z 514.745,A -85,B 0,C 180,E1 -17578.992,E2 -17578.992} C_VEL
LIN {X 0,Y 431.522,Z 502.652,A -85,B 0,C 180,E1 -17580.208,E2 -17580.208} C_VEL
LIN {X 0,Y 432.908,Z 490.693,A -85,B 0,C 180,E1 -17581.179,E2 -17581.179} C_VEL
LIN {X 0,Y 434.188,Z 477.53,A -85,B 0,C 180,E1 -17582.026,E2 -17582.026} C_VEL
LIN {X 0,Y 435.03,Z 465.261,A -85,B 0,C 180,E1 -17582.639,E2 -17582.639} C_VEL
LIN {X 0,Y 435.791,Z 451.111,A -85,B 0,C 180,E1 -17583.152,E2 -17583.152} C_VEL
LIN {X 0,Y 436.273,Z 436.534,A -85,B 0,C 180,E1 -17583.48,E2 -17583.48} C_VEL
LIN {X 0,Y 438.422,Z 342.874,A -85,B 0,C 180,E1 -17585.036,E2 -17585.036} C_VEL
LIN {X 0,Y 429.867,Z 322.908,A -85,B 0,C 180,E1 -17586.001,E2 -17586.001} C_VEL
LIN {X 0,Y 423.461,Z 309.415,A -85,B 0,C 180,E1 -17586.749,E2 -17586.749} C_VEL
LIN {X 0,Y 422.335,Z 304.431,A -85,B 0,C 180,E1 -17588.151,E2 -17588.151} C_VEL
LIN {X 0,Y 422.305,Z 304.43,A -85,B 0,C 180,E1 -17591.559,E2 -17591.559} C_VEL
LIN {X 0,Y 422.344,Z 304.42,A -85,B 0,C 180,E1 -17594.509,E2 -17594.509} C_VEL
LIN {X 0,Y 422.317,Z 304.437,A -85,B 0,C 180,E1 -17597.155,E2 -17597.155} C_VEL
LIN {X 0,Y 422.356,Z 304.432,A -85,B 0,C 180,E1 -17599.714,E2 -17599.714} C_VEL
LIN {X 0,Y 422.34,Z 304.415,A -85,B 0,C 180,E1 -17603.341,E2 -17603.341} C_VEL
LIN {X 0,Y 422.366,Z 304.419,A -85,B 0,C 180,E1 -17606.01,E2 -17606.01} C_VEL
LIN {X 0,Y 422.362,Z 304.426,A -85,B 0,C 180,E1 -17609.577,E2 -17609.577} C_VEL
LIN {X 0,Y 422.38,Z 304.419,A -85,B 0,C 180,E1 -17612.333,E2 -17612.333} C_VEL
LIN {X 0,Y 422.376,Z 304.423,A -85,B 0,C 180,E1 -17615.788,E2 -17615.788} C_VEL
LIN {X 0,Y 422.402,Z 304.424,A -85,B 0,C 180,E1 -17618.604,E2 -17618.604} C_VEL
LIN {X 0,Y 422.406,Z 304.417,A -85,B 0,C 180,E1 -17621.635,E2 -17621.635} C_VEL
LIN {X 0,Y 422.446,Z 304.417,A -85,B 0,C 180,E1 -17624.616,E2 -17624.616} C_VEL
LIN {X 0,Y 422.543,Z 304.407,A -85,B 0,C 180,E1 -17628.526,E2 -17628.526} C_VEL
LIN {X 0,Y 422.59,Z 304.396,A -85,B 0,C 180,E1 -17632.38,E2 -17632.38} C_VEL
LIN {X 0,Y 422.689,Z 304.381,A -85,B 0,C 180,E1 -17635.247,E2 -17635.247} C_VEL
LIN {X 0,Y 422.524,Z 304.407,A -85,B 0,C 180,E1 -17638.1,E2 -17638.1} C_VEL
LIN {X 0,Y 422.666,Z 304.389,A -85,B 0,C 180,E1 -17640,E2 -17640} C_VEL
LIN {X 0,Y 422.658,Z 304.391,A -85,B 0,C 180,E1 -17643.801,E2 -17643.801} C_VEL
LIN {X 0,Y 422.615,Z 304.388,A -85,B 0,C 180,E1 -17646.662,E2 -17646.662} C_VEL
LIN {X 0,Y 422.547,Z 304.405,A -85,B 0,C 180,E1 -17649.542,E2 -17649.542} C_VEL
LIN {X 0,Y 422.516,Z 304.397,A -85,B 0,C 180,E1 -17652.446,E2 -17652.446} C_VEL
LIN {X 0,Y 422.462,Z 304.413,A -85,B 0,C 180,E1 -17655.932,E2 -17655.932} C_VEL
LIN {X 0,Y 422.424,Z 304.421,A -85,B 0,C 180,E1 -17659.368,E2 -17659.368} C_VEL
LIN {X 0,Y 422.379,Z 304.417,A -85,B 0,C 180,E1 -17662.421,E2 -17662.421} C_VEL
LIN {X 0,Y 422.369,Z 304.425,A -85,B 0,C 180,E1 -17665.542,E2 -17665.542} C_VEL
LIN {X 0,Y 422.377,Z 304.43,A -85,B 0,C 180,E1 -17668.745,E2 -17668.745} C_VEL
LIN {X 0,Y 422.39,Z 304.429,A -85,B 0,C 180,E1 -17672.256,E2 -17672.256} C_VEL
LIN {X 0,Y 422.413,Z 304.391,A -85,B 0,C 180,E1 -17675.663,E2 -17675.663} C_VEL
LIN {X 0,Y 422.417,Z 304.423,A -85,B 0,C 180,E1 -17679.058,E2 -17679.058} C_VEL
LIN {X 0,Y 422.346,Z 304.434,A -85,B 0,C 180,E1 -17681.733,E2 -17681.733} C_VEL
LIN {X 0,Y 422.36,Z 304.43,A -85,B 0,C 180,E1 -17684.515,E2 -17684.515} C_VEL
LIN {X 0,Y 422.374,Z 304.427,A -85,B 0,C 180,E1 -17687.166,E2 -17687.166} C_VEL
LIN {X 0,Y 422.41,Z 304.424,A -85,B 0,C 180,E1 -17690.945,E2 -17690.945} C_VEL
LIN {X 0,Y 422.42,Z 304.422,A -85,B 0,C 180,E1 -17694.341,E2 -17694.341} C_VEL
LIN {X 0,Y 422.428,Z 304.543,A -85,B 0,C 180,E1 -17695.764,E2 -17695.764} C_VEL
LIN {X 0,Y 425.534,Z 316.935,A -85,B 0,C 180,E1 -17698.611,E2 -17698.611} C_VEL
LIN {X 0,Y 428.491,Z 330.005,A -85,B 0,C 180,E1 -17701.439,E2 -17701.439} C_VEL
LIN {X 0,Y 430.068,Z 338.3,A -85,B 0,C 180,E1 -17703.154,E2 -17703.154} C_VEL
LIN {X 0,Y 428.186,Z 352.301,A -85,B 0,C 180,E1 -17705.676,E2 -17705.676} C_VEL
LIN {X 0,Y 433.494,Z 380.188,A -85,B 0,C 180,E1 -17706.559,E2 -17706.559} C_VEL
LIN {X 0,Y 437.069,Z 404.247,A -85,B 0,C 180,E1 -17707.232,E2 -17707.232} C_VEL
LIN {X 0,Y 435.632,Z 468.419,A -85,B 0,C 180,E1 -17708.299,E2 -17708.299} C_VEL
LIN {X 0,Y 435.047,Z 492.315,A -85,B 0,C 180,E1 -17708.733,E2 -17708.733} C_VEL
LIN {X 0,Y 434.04,Z 507.072,A -85,B 0,C 180,E1 -17709.177,E2 -17709.177} C_VEL
LIN {X 0,Y 432.637,Z 521.396,A -85,B 0,C 180,E1 -17709.804,E2 -17709.804} C_VEL
LIN {X 0,Y 431.201,Z 534.397,A -85,B 0,C 180,E1 -17710.575,E2 -17710.575} C_VEL
LIN {X 0,Y 429.493,Z 547.651,A -85,B 0,C 180,E1 -17711.583,E2 -17711.583} C_VEL
LIN {X 0,Y 427.718,Z 559.703,A -85,B 0,C 180,E1 -17712.736,E2 -17712.736} C_VEL
LIN {X 0,Y 425.918,Z 570.602,A -85,B 0,C 180,E1 -17714.013,E2 -17714.013} C_VEL
LIN {X 0,Y 424.361,Z 580.444,A -85,B 0,C 180,E1 -17715.424,E2 -17715.424} C_VEL
LIN {X 0,Y 423.009,Z 589.885,A -85,B 0,C 180,E1 -17717.085,E2 -17717.085} C_VEL
LIN {X 0,Y 421.899,Z 597.555,A -85,B 0,C 180,E1 -17718.753,E2 -17718.753} C_VEL
LIN {X 0,Y 421.065,Z 603.737,A -85,B 0,C 180,E1 -17720.427,E2 -17720.427} C_VEL
LIN {X 0,Y 420.445,Z 609.251,A -85,B 0,C 180,E1 -17722.343,E2 -17722.343} C_VEL
LIN {X 0,Y 420.349,Z 613.294,A -85,B 0,C 180,E1 -17724.264,E2 -17724.264} C_VEL
LIN {X 0,Y 420.266,Z 617.432,A -85,B 0,C 180,E1 -17725.701,E2 -17725.701} C_VEL
LIN {X 0,Y 420.271,Z 620.576,A -85,B 0,C 180,E1 -17727.136,E2 -17727.136} C_VEL
LIN {X 0,Y 420.286,Z 623.428,A -85,B 0,C 180,E1 -17729.047,E2 -17729.047} C_VEL
LIN {X 0,Y 420.245,Z 624.78,A -85,B 0,C 180,E1 -17730.957,E2 -17730.957} C_VEL
LIN {X 0,Y 420.183,Z 624.639,A -85,B 0,C 180,E1 -17732.869,E2 -17732.869} C_VEL
LIN {X 0,Y 420.267,Z 623.048,A -85,B 0,C 180,E1 -17734.782,E2 -17734.782} C_VEL
LIN {X 0,Y 420.515,Z 620.007,A -85,B 0,C 180,E1 -17736.698,E2 -17736.698} C_VEL
LIN {X 0,Y 420.984,Z 615.44,A -85,B 0,C 180,E1 -17738.614,E2 -17738.614} C_VEL
LIN {X 0,Y 421.721,Z 610.929,A -85,B 0,C 180,E1 -17740.046,E2 -17740.046} C_VEL
LIN {X 0,Y 422.8,Z 604.065,A -85,B 0,C 180,E1 -17741.784,E2 -17741.784} C_VEL
LIN {X 0,Y 424.037,Z 596.25,A -85,B 0,C 180,E1 -17743.373,E2 -17743.373} C_VEL
LIN {X 0,Y 425.434,Z 587.8,A -85,B 0,C 180,E1 -17744.787,E2 -17744.787} C_VEL
LIN {X 0,Y 427.071,Z 577.665,A -85,B 0,C 180,E1 -17746.192,E2 -17746.192} C_VEL
LIN {X 0,Y 428.795,Z 566.432,A -85,B 0,C 180,E1 -17747.469,E2 -17747.469} C_VEL
LIN {X 0,Y 430.593,Z 554.037,A -85,B 0,C 180,E1 -17748.619,E2 -17748.619} C_VEL
LIN {X 0,Y 432.231,Z 541.928,A -85,B 0,C 180,E1 -17749.528,E2 -17749.528} C_VEL
LIN {X 0,Y 433.81,Z 528.149,A -85,B 0,C 180,E1 -17750.357,E2 -17750.357} C_VEL
LIN {X 0,Y 435.334,Z 513.63,A -85,B 0,C 180,E1 -17751.01,E2 -17751.01} C_VEL
LIN {X 0,Y 436.502,Z 498.879,A -85,B 0,C 180,E1 -17751.475,E2 -17751.475} C_VEL
LIN {X 0,Y 441.342,Z 405.317,A -85,B 0,C 180,E1 -17753.717,E2 -17753.717} C_VEL
LIN {X 0,Y 440.113,Z 389.648,A -85,B 0,C 180,E1 -17754.305,E2 -17754.305} C_VEL
LIN {X 0,Y 437.352,Z 367.99,A -85,B 0,C 180,E1 -17755.256,E2 -17755.256} C_VEL
LIN {X 0,Y 434.828,Z 353.353,A -85,B 0,C 180,E1 -17756.022,E2 -17756.022} C_VEL
LIN {X 0,Y 433.92,Z 339.82,A -85,B 0,C 180,E1 -17757.163,E2 -17757.163} C_VEL
LIN {X 0,Y 432.663,Z 333.576,A -85,B 0,C 180,E1 -17757.845,E2 -17757.845} C_VEL
LIN {X 0,Y 429.308,Z 320.683,A -85,B 0,C 180,E1 -17759.485,E2 -17759.485} C_VEL
LIN {X 0,Y 427.115,Z 313.533,A -85,B 0,C 180,E1 -17760.558,E2 -17760.558} C_VEL
LIN {X 0,Y 424.08,Z 308.246,A -85,B 0,C 180,E1 -17761.674,E2 -17761.674} C_VEL
LIN {X 0,Y 422.564,Z 305.559,A -85,B 0,C 180,E1 -17762.287,E2 -17762.287} C_VEL
LIN {X 0,Y 422.327,Z 304.429,A -85,B 0,C 180,E1 -17762.504,E2 -17762.504} C_VEL
LIN {X 0,Y 422.321,Z 304.437,A -85,B 0,C 180,E1 -17765.64,E2 -17765.64} C_VEL
LIN {X 0,Y 422.32,Z 304.438,A -85,B 0,C 180,E1 -17768.783,E2 -17768.783} C_VEL
LIN {X 0,Y 422.322,Z 304.436,A -85,B 0,C 180,E1 -17771.725,E2 -17771.725} C_VEL
LIN {X 0,Y 422.365,Z 304.43,A -85,B 0,C 180,E1 -17774.512,E2 -17774.512} C_VEL
LIN {X 0,Y 422.33,Z 304.434,A -85,B 0,C 180,E1 -17777.157,E2 -17777.157} C_VEL
LIN {X 0,Y 422.359,Z 304.43,A -85,B 0,C 180,E1 -17779.72,E2 -17779.72} C_VEL
LIN {X 0,Y 422.362,Z 304.432,A -85,B 0,C 180,E1 -17783.343,E2 -17783.343} C_VEL
LIN {X 0,Y 422.394,Z 304.426,A -85,B 0,C 180,E1 -17786.013,E2 -17786.013} C_VEL
LIN {X 0,Y 422.382,Z 304.43,A -85,B 0,C 180,E1 -17789.582,E2 -17789.582} C_VEL
LIN {X 0,Y 422.406,Z 304.428,A -85,B 0,C 180,E1 -17792.335,E2 -17792.335} C_VEL
LIN {X 0,Y 422.422,Z 304.43,A -85,B 0,C 180,E1 -17796.036,E2 -17796.036} C_VEL
LIN {X 0,Y 422.439,Z 304.67,A -85,B 0,C 180,E1 -17796.175,E2 -17796.175} C_VEL
LIN {X 0,Y 426.205,Z 314.081,A -85,B 0,C 180,E1 -17798.804,E2 -17798.804} C_VEL
LIN {X 0,Y 429.757,Z 324.449,A -85,B 0,C 180,E1 -17801.362,E2 -17801.362} C_VEL
LIN {X 0,Y 433.038,Z 336.55,A -85,B 0,C 180,E1 -17804.039,E2 -17804.039} C_VEL
LIN {X 0,Y 434.843,Z 346.65,A -85,B 0,C 180,E1 -17806.049,E2 -17806.049} C_VEL
LIN {X 0,Y 438.54,Z 360.955,A -85,B 0,C 180,E1 -17806.906,E2 -17806.906} C_VEL
LIN {X 0,Y 441.908,Z 378.477,A -85,B 0,C 180,E1 -17807.784,E2 -17807.784} C_VEL
LIN {X 0,Y 442.78,Z 383.941,A -85,B 0,C 180,E1 -17808.032,E2 -17808.032} C_VEL
LIN {X 0,Y 437.116,Z 488.087,A -85,B 0,C 180,E1 -17810.517,E2 -17810.517} C_VEL
LIN {X 0,Y 435.961,Z 502.455,A -85,B 0,C 180,E1 -17811.046,E2 -17811.046} C_VEL
LIN {X 0,Y 434.561,Z 516.862,A -85,B 0,C 180,E1 -17811.776,E2 -17811.776} C_VEL
LIN {X 0,Y 432.91,Z 530.681,A -85,B 0,C 180,E1 -17812.68,E2 -17812.68} C_VEL
LIN {X 0,Y 431.166,Z 543.153,A -85,B 0,C 180,E1 -17813.704,E2 -17813.704} C_VEL
LIN {X 0,Y 429.478,Z 554.653,A -85,B 0,C 180,E1 -17814.872,E2 -17814.872} C_VEL
LIN {X 0,Y 427.745,Z 565.731,A -85,B 0,C 180,E1 -17816.244,E2 -17816.244} C_VEL
LIN {X 0,Y 426.111,Z 575.105,A -85,B 0,C 180,E1 -17817.645,E2 -17817.645} C_VEL
LIN {X 0,Y 424.345,Z 584.135,A -85,B 0,C 180,E1 -17819.291,E2 -17819.291} C_VEL
LIN {X 0,Y 423.052,Z 591.355,A -85,B 0,C 180,E1 -17820.949,E2 -17820.949} C_VEL
LIN {X 0,Y 421.93,Z 597.843,A -85,B 0,C 180,E1 -17822.855,E2 -17822.855} C_VEL
LIN {X 0,Y 421.262,Z 602.655,A -85,B 0,C 180,E1 -17824.769,E2 -17824.769} C_VEL
LIN {X 0,Y 420.639,Z 605.957,A -85,B 0,C 180,E1 -17826.694,E2 -17826.694} C_VEL
LIN {X 0,Y 420.255,Z 607.749,A -85,B 0,C 180,E1 -17828.627,E2 -17828.627} C_VEL
LIN {X 0,Y 420.137,Z 608.092,A -85,B 0,C 180,E1 -17830.567,E2 -17830.567} C_VEL
LIN {X 0,Y 419.968,Z 606.963,A -85,B 0,C 180,E1 -17832.522,E2 -17832.522} C_VEL
LIN {X 0,Y 420.087,Z 604.323,A -85,B 0,C 180,E1 -17834.484,E2 -17834.484} C_VEL
LIN {X 0,Y 420.149,Z 601.232,A -85,B 0,C 180,E1 -17835.967,E2 -17835.967} C_VEL
LIN {X 0,Y 420.344,Z 597.171,A -85,B 0,C 180,E1 -17837.454,E2 -17837.454} C_VEL
LIN {X 0,Y 420.586,Z 592.02,A -85,B 0,C 180,E1 -17838.951,E2 -17838.951} C_VEL
LIN {X 0,Y 420.981,Z 584.437,A -85,B 0,C 180,E1 -17840.706,E2 -17840.706} C_VEL
LIN {X 0,Y 421.48,Z 576.376,A -85,B 0,C 180,E1 -17842.215,E2 -17842.215} C_VEL
LIN {X 0,Y 422.114,Z 566.857,A -85,B 0,C 180,E1 -17843.686,E2 -17843.686} C_VEL
LIN {X 0,Y 422.752,Z 556.647,A -85,B 0,C 180,E1 -17844.993,E2 -17844.993} C_VEL
LIN {X 0,Y 423.64,Z 544.675,A -85,B 0,C 180,E1 -17846.25,E2 -17846.25} C_VEL
LIN {X 0,Y 424.455,Z 532.077,A -85,B 0,C 180,E1 -17847.331,E2 -17847.331} C_VEL
LIN {X 0,Y 425.202,Z 518.52,A -85,B 0,C 180,E1 -17848.269,E2 -17848.269} C_VEL
LIN {X 0,Y 425.985,Z 504.49,A -85,B 0,C 180,E1 -17849.017,E2 -17849.017} C_VEL
LIN {X 0,Y 426.713,Z 489.387,A -85,B 0,C 180,E1 -17849.603,E2 -17849.603} C_VEL
LIN {X 0,Y 427.168,Z 473.712,A -85,B 0,C 180,E1 -17850.008,E2 -17850.008} C_VEL
LIN {X 0,Y 429.488,Z 375.997,A -85,B 0,C 180,E1 -17852.106,E2 -17852.106} C_VEL
LIN {X 0,Y 425.508,Z 344.391,A -85,B 0,C 180,E1 -17852.96,E2 -17852.96} C_VEL
LIN {X 0,Y 426.443,Z 326.819,A -85,B 0,C 180,E1 -17855.669,E2 -17855.669} C_VEL
LIN {X 0,Y 426.08,Z 322.667,A -85,B 0,C 180,E1 -17856.337,E2 -17856.337} C_VEL
LIN {X 0,Y 422.37,Z 304.431,A -85,B 0,C 180,E1 -17859.389,E2 -17859.389} C_VEL
LIN {X 0,Y 422.358,Z 304.428,A -85,B 0,C 180,E1 -17863.136,E2 -17863.136} C_VEL
LIN {X 0,Y 422.368,Z 304.428,A -85,B 0,C 180,E1 -17865.849,E2 -17865.849} C_VEL
LIN {X 0,Y 422.336,Z 304.432,A -85,B 0,C 180,E1 -17869.721,E2 -17869.721} C_VEL
LIN {X 0,Y 422.338,Z 304.43,A -85,B 0,C 180,E1 -17873.338,E2 -17873.338} C_VEL
LIN {X 0,Y 422.318,Z 304.433,A -85,B 0,C 180,E1 -17876.814,E2 -17876.814} C_VEL
LIN {X 0,Y 422.356,Z 304.435,A -85,B 0,C 180,E1 -17880.161,E2 -17880.161} C_VEL
LIN {X 0,Y 422.387,Z 304.425,A -85,B 0,C 180,E1 -17883.57,E2 -17883.57} C_VEL
LIN {X 0,Y 422.395,Z 304.425,A -85,B 0,C 180,E1 -17886.546,E2 -17886.546} C_VEL
LIN {X 0,Y 422.409,Z 304.425,A -85,B 0,C 180,E1 -17889.619,E2 -17889.619} C_VEL
LIN {X 0,Y 422.427,Z 304.42,A -85,B 0,C 180,E1 -17892.632,E2 -17892.632} C_VEL
LIN {X 0,Y 422.481,Z 304.417,A -85,B 0,C 180,E1 -17895.598,E2 -17895.598} C_VEL
LIN {X 0,Y 422.571,Z 304.403,A -85,B 0,C 180,E1 -17898.525,E2 -17898.525} C_VEL
LIN {X 0,Y 422.505,Z 304.442,A -85,B 0,C 180,E1 -17899.732,E2 -17899.732} C_VEL
LIN {X 0,Y 423.29,Z 308.188,A -85,B 0,C 180,E1 -17900.6,E2 -17900.6} C_VEL
LIN {X 0,Y 429.856,Z 328.846,A -85,B 0,C 180,E1 -17901.24,E2 -17901.24} C_VEL
LIN {X 0,Y 431.124,Z 335.825,A -85,B 0,C 180,E1 -17901.413,E2 -17901.413} C_VEL
LIN {X 0,Y 429.127,Z 443.23,A -85,B 0,C 180,E1 -17903.202,E2 -17903.202} C_VEL
LIN {X 0,Y 428.692,Z 457.842,A -85,B 0,C 180,E1 -17903.636,E2 -17903.636} C_VEL
LIN {X 0,Y 428.099,Z 471.742,A -85,B 0,C 180,E1 -17904.246,E2 -17904.246} C_VEL
LIN {X 0,Y 427.264,Z 485.559,A -85,B 0,C 180,E1 -17905.06,E2 -17905.06} C_VEL
LIN {X 0,Y 426.56,Z 496.499,A -85,B 0,C 180,E1 -17905.878,E2 -17905.878} C_VEL
LIN {X 0,Y 425.359,Z 508.138,A -85,B 0,C 180,E1 -17906.93,E2 -17906.93} C_VEL
LIN {X 0,Y 424.584,Z 518.704,A -85,B 0,C 180,E1 -17908.107,E2 -17908.107} C_VEL
LIN {X 0,Y 423.521,Z 529.238,A -85,B 0,C 180,E1 -17909.524,E2 -17909.524} C_VEL
LIN {X 0,Y 422.709,Z 537.926,A -85,B 0,C 180,E1 -17910.947,E2 -17910.947} C_VEL
LIN {X 0,Y 421.932,Z 545.176,A -85,B 0,C 180,E1 -17912.376,E2 -17912.376} C_VEL
LIN {X 0,Y 421.569,Z 552,A -85,B 0,C 180,E1 -17914.026,E2 -17914.026} C_VEL
LIN {X 0,Y 421.092,Z 557.608,A -85,B 0,C 180,E1 -17915.725,E2 -17915.725} C_VEL
LIN {X 0,Y 420.681,Z 562.424,A -85,B 0,C 180,E1 -17917.652,E2 -17917.652} C_VEL
LIN {X 0,Y 420.502,Z 565.748,A -85,B 0,C 180,E1 -17919.586,E2 -17919.586} C_VEL
LIN {X 0,Y 420.438,Z 567.665,A -85,B 0,C 180,E1 -17921.53,E2 -17921.53} C_VEL
LIN {X 0,Y 420.532,Z 568.229,A -85,B 0,C 180,E1 -17923.482,E2 -17923.482} C_VEL
LIN {X 0,Y 420.823,Z 567.436,A -85,B 0,C 180,E1 -17925.442,E2 -17925.442} C_VEL
LIN {X 0,Y 421.203,Z 565.26,A -85,B 0,C 180,E1 -17927.415,E2 -17927.415} C_VEL
LIN {X 0,Y 421.92,Z 561.618,A -85,B 0,C 180,E1 -17929.389,E2 -17929.389} C_VEL
LIN {X 0,Y 422.905,Z 556.391,A -85,B 0,C 180,E1 -17931.367,E2 -17931.367} C_VEL
LIN {X 0,Y 424.001,Z 550.059,A -85,B 0,C 180,E1 -17933.154,E2 -17933.154} C_VEL
LIN {X 0,Y 423.865,Z 547.304,A -85,B 0,C 180,E1 -17933.86,E2 -17933.86} C_VEL
LIN {X 0,Y 421.985,Z 542.607,A -85,B 0,C 180,E1 -17935.019,E2 -17935.019} C_VEL
LIN {X 0,Y 420.193,Z 537.429,A -85,B 0,C 180,E1 -17936.143,E2 -17936.143} C_VEL
LIN {X 0,Y 420.186,Z 533.847,A -85,B 0,C 180,E1 -17936.785,E2 -17936.785} C_VEL
LIN {X 0,Y 421.717,Z 525.164,A -85,B 0,C 180,E1 -17938.084,E2 -17938.084} C_VEL
LIN {X 0,Y 423.437,Z 513.89,A -85,B 0,C 180,E1 -17939.477,E2 -17939.477} C_VEL
LIN {X 0,Y 425.001,Z 502.867,A -85,B 0,C 180,E1 -17940.584,E2 -17940.584} C_VEL
LIN {X 0,Y 426.5,Z 490.273,A -85,B 0,C 180,E1 -17941.613,E2 -17941.613} C_VEL
LIN {X 0,Y 427.831,Z 476.54,A -85,B 0,C 180,E1 -17942.49,E2 -17942.49} C_VEL
LIN {X 0,Y 428.748,Z 463.866,A -85,B 0,C 180,E1 -17943.108,E2 -17943.108} C_VEL
LIN {X 0,Y 429.508,Z 449.647,A -85,B 0,C 180,E1 -17943.6,E2 -17943.6} C_VEL
LIN {X 0,Y 429.919,Z 433.232,A -85,B 0,C 180,E1 -17943.95,E2 -17943.95} C_VEL
LIN {X 0,Y 432.037,Z 344.564,A -85,B 0,C 180,E1 -17945.444,E2 -17945.444} C_VEL
LIN {X 0,Y 423.102,Z 323.921,A -85,B 0,C 180,E1 -17946.479,E2 -17946.479} C_VEL
LIN {X 0,Y 416.372,Z 309.938,A -85,B 0,C 180,E1 -17947.269,E2 -17947.269} C_VEL
LIN {X 0,Y 415.281,Z 305.307,A -85,B 0,C 180,E1 -17948.61,E2 -17948.61} C_VEL
LIN {X 0,Y 415.262,Z 305.309,A -85,B 0,C 180,E1 -17952.083,E2 -17952.083} C_VEL
LIN {X 0,Y 415.286,Z 305.297,A -85,B 0,C 180,E1 -17955.1,E2 -17955.1} C_VEL
LIN {X 0,Y 415.267,Z 305.313,A -85,B 0,C 180,E1 -17957.911,E2 -17957.911} C_VEL
LIN {X 0,Y 415.295,Z 305.312,A -85,B 0,C 180,E1 -17961.388,E2 -17961.388} C_VEL
LIN {X 0,Y 415.316,Z 305.284,A -85,B 0,C 180,E1 -17965.011,E2 -17965.011} C_VEL
LIN {X 0,Y 415.301,Z 305.305,A -85,B 0,C 180,E1 -17968.477,E2 -17968.477} C_VEL
LIN {X 0,Y 415.328,Z 305.302,A -85,B 0,C 180,E1 -17971.822,E2 -17971.822} C_VEL
LIN {X 0,Y 415.32,Z 305.309,A -85,B 0,C 180,E1 -17975.063,E2 -17975.063} C_VEL
LIN {X 0,Y 415.366,Z 305.302,A -85,B 0,C 180,E1 -17978.223,E2 -17978.223} C_VEL
LIN {X 0,Y 415.368,Z 305.292,A -85,B 0,C 180,E1 -17981.313,E2 -17981.313} C_VEL
LIN {X 0,Y 415.39,Z 305.296,A -85,B 0,C 180,E1 -17984.348,E2 -17984.348} C_VEL
LIN {X 0,Y 415.51,Z 305.285,A -85,B 0,C 180,E1 -17987.87,E2 -17987.87} C_VEL
LIN {X 0,Y 415.52,Z 305.27,A -85,B 0,C 180,E1 -17991.274,E2 -17991.274} C_VEL
LIN {X 0,Y 415.624,Z 305.268,A -85,B 0,C 180,E1 -17994.197,E2 -17994.197} C_VEL
LIN {X 0,Y 415.601,Z 305.26,A -85,B 0,C 180,E1 -17997.102,E2 -17997.102} C_VEL
LIN {X 0,Y 415.62,Z 305.267,A -85,B 0,C 180,E1 -18000,E2 -18000} C_VEL
LIN {X 0,Y 415.624,Z 305.267,A -85,B 0,C 180,E1 -18003.865,E2 -18003.865} C_VEL
LIN {X 0,Y 415.577,Z 305.263,A -85,B 0,C 180,E1 -18006.776,E2 -18006.776} C_VEL
LIN {X 0,Y 415.501,Z 305.282,A -85,B 0,C 180,E1 -18009.705,E2 -18009.705} C_VEL
LIN {X 0,Y 415.454,Z 305.276,A -85,B 0,C 180,E1 -18012.661,E2 -18012.661} C_VEL
LIN {X 0,Y 415.426,Z 305.29,A -85,B 0,C 180,E1 -18016.052,E2 -18016.052} C_VEL
LIN {X 0,Y 415.362,Z 305.299,A -85,B 0,C 180,E1 -18019.711,E2 -18019.711} C_VEL
LIN {X 0,Y 415.314,Z 305.3,A -85,B 0,C 180,E1 -18022.824,E2 -18022.824} C_VEL
LIN {X 0,Y 415.324,Z 305.301,A -85,B 0,C 180,E1 -18026.008,E2 -18026.008} C_VEL
LIN {X 0,Y 415.328,Z 305.304,A -85,B 0,C 180,E1 -18029.28,E2 -18029.28} C_VEL
LIN {X 0,Y 415.321,Z 305.308,A -85,B 0,C 180,E1 -18032.662,E2 -18032.662} C_VEL
LIN {X 0,Y 415.386,Z 305.268,A -85,B 0,C 180,E1 -18036.17,E2 -18036.17} C_VEL
LIN {X 0,Y 415.378,Z 305.3,A -85,B 0,C 180,E1 -18039.137,E2 -18039.137} C_VEL
LIN {X 0,Y 415.305,Z 305.308,A -85,B 0,C 180,E1 -18042.426,E2 -18042.426} C_VEL
LIN {X 0,Y 415.329,Z 305.302,A -85,B 0,C 180,E1 -18045.099,E2 -18045.099} C_VEL
LIN {X 0,Y 415.319,Z 305.307,A -85,B 0,C 180,E1 -18047.908,E2 -18047.908} C_VEL
LIN {X 0,Y 415.373,Z 305.301,A -85,B 0,C 180,E1 -18051.4,E2 -18051.4} C_VEL
LIN {X 0,Y 415.392,Z 305.294,A -85,B 0,C 180,E1 -18054.036,E2 -18054.036} C_VEL
LIN {X 0,Y 415.362,Z 305.379,A -85,B 0,C 180,E1 -18055.264,E2 -18055.264} C_VEL
LIN {X 0,Y 418.518,Z 317.655,A -85,B 0,C 180,E1 -18058.162,E2 -18058.162} C_VEL
LIN {X 0,Y 421.284,Z 329.975,A -85,B 0,C 180,E1 -18060.904,E2 -18060.904} C_VEL
LIN {X 0,Y 423.183,Z 339.567,A -85,B 0,C 180,E1 -18062.927,E2 -18062.927} C_VEL
LIN {X 0,Y 422.196,Z 347.771,A -85,B 0,C 180,E1 -18064.45,E2 -18064.45} C_VEL
LIN {X 0,Y 421.556,Z 351.798,A -85,B 0,C 180,E1 -18065.183,E2 -18065.183} C_VEL
LIN {X 0,Y 427.109,Z 380.94,A -85,B 0,C 180,E1 -18066.135,E2 -18066.135} C_VEL
LIN {X 0,Y 430.677,Z 404.791,A -85,B 0,C 180,E1 -18066.823,E2 -18066.823} C_VEL
LIN {X 0,Y 429.306,Z 466.117,A -85,B 0,C 180,E1 -18067.859,E2 -18067.859} C_VEL
LIN {X 0,Y 428.634,Z 492.109,A -85,B 0,C 180,E1 -18068.336,E2 -18068.336} C_VEL
LIN {X 0,Y 427.579,Z 506.799,A -85,B 0,C 180,E1 -18068.784,E2 -18068.784} C_VEL
LIN {X 0,Y 426.236,Z 520.22,A -85,B 0,C 180,E1 -18069.376,E2 -18069.376} C_VEL
LIN {X 0,Y 424.784,Z 533.224,A -85,B 0,C 180,E1 -18070.147,E2 -18070.147} C_VEL
LIN {X 0,Y 423.18,Z 545.206,A -85,B 0,C 180,E1 -18071.047,E2 -18071.047} C_VEL
LIN {X 0,Y 421.292,Z 557.703,A -85,B 0,C 180,E1 -18072.214,E2 -18072.214} C_VEL
LIN {X 0,Y 419.365,Z 568.893,A -85,B 0,C 180,E1 -18073.507,E2 -18073.507} C_VEL
LIN {X 0,Y 417.737,Z 578.947,A -85,B 0,C 180,E1 -18074.939,E2 -18074.939} C_VEL
LIN {X 0,Y 416.405,Z 587.334,A -85,B 0,C 180,E1 -18076.382,E2 -18076.382} C_VEL
LIN {X 0,Y 415.18,Z 595.489,A -85,B 0,C 180,E1 -18078.1,E2 -18078.1} C_VEL
LIN {X 0,Y 414.213,Z 601.91,A -85,B 0,C 180,E1 -18079.775,E2 -18079.775} C_VEL
LIN {X 0,Y 413.506,Z 607.742,A -85,B 0,C 180,E1 -18081.724,E2 -18081.724} C_VEL
LIN {X 0,Y 413.305,Z 611.129,A -85,B 0,C 180,E1 -18083.189,E2 -18083.189} C_VEL
LIN {X 0,Y 413.254,Z 613.43,A -85,B 0,C 180,E1 -18084.41,E2 -18084.41} C_VEL
LIN {X 0,Y 413.166,Z 618.073,A -85,B 0,C 180,E1 -18086.114,E2 -18086.114} C_VEL
LIN {X 0,Y 413.204,Z 620.141,A -85,B 0,C 180,E1 -18087.087,E2 -18087.087} C_VEL
LIN {X 0,Y 413.206,Z 623.1,A -85,B 0,C 180,E1 -18089.031,E2 -18089.031} C_VEL
LIN {X 0,Y 413.171,Z 624.556,A -85,B 0,C 180,E1 -18090.974,E2 -18090.974} C_VEL
LIN {X 0,Y 413.091,Z 624.545,A -85,B 0,C 180,E1 -18092.918,E2 -18092.918} C_VEL
LIN {X 0,Y 413.194,Z 623.066,A -85,B 0,C 180,E1 -18094.865,E2 -18094.865} C_VEL
LIN {X 0,Y 413.449,Z 620.126,A -85,B 0,C 180,E1 -18096.813,E2 -18096.813} C_VEL
LIN {X 0,Y 413.956,Z 615.68,A -85,B 0,C 180,E1 -18098.762,E2 -18098.762} C_VEL
LIN {X 0,Y 415.076,Z 609.589,A -85,B 0,C 180,E1 -18100.7,E2 -18100.7} C_VEL
LIN {X 0,Y 415.948,Z 603.599,A -85,B 0,C 180,E1 -18102.208,E2 -18102.208} C_VEL
LIN {X 0,Y 417.383,Z 595.624,A -85,B 0,C 180,E1 -18103.838,E2 -18103.838} C_VEL
LIN {X 0,Y 418.927,Z 587.079,A -85,B 0,C 180,E1 -18105.27,E2 -18105.27} C_VEL
LIN {X 0,Y 420.589,Z 576.864,A -85,B 0,C 180,E1 -18106.697,E2 -18106.697} C_VEL
LIN {X 0,Y 422.505,Z 565.478,A -85,B 0,C 180,E1 -18107.987,E2 -18107.987} C_VEL
LIN {X 0,Y 424.403,Z 552.97,A -85,B 0,C 180,E1 -18109.151,E2 -18109.151} C_VEL
LIN {X 0,Y 426.36,Z 539.065,A -85,B 0,C 180,E1 -18110.184,E2 -18110.184} C_VEL
LIN {X 0,Y 427.901,Z 526.039,A -85,B 0,C 180,E1 -18110.941,E2 -18110.941} C_VEL
LIN {X 0,Y 429.525,Z 510.256,A -85,B 0,C 180,E1 -18111.621,E2 -18111.621} C_VEL
LIN {X 0,Y 430.704,Z 495.413,A -85,B 0,C 180,E1 -18112.062,E2 -18112.062} C_VEL
LIN {X 0,Y 435.58,Z 406.323,A -85,B 0,C 180,E1 -18114.241,E2 -18114.241} C_VEL
LIN {X 0,Y 434.349,Z 390.28,A -85,B 0,C 180,E1 -18114.865,E2 -18114.865} C_VEL
LIN {X 0,Y 431.827,Z 370.09,A -85,B 0,C 180,E1 -18115.784,E2 -18115.784} C_VEL
LIN {X 0,Y 429.023,Z 353.523,A -85,B 0,C 180,E1 -18116.671,E2 -18116.671} C_VEL
LIN {X 0,Y 428.328,Z 341.765,A -85,B 0,C 180,E1 -18117.714,E2 -18117.714} C_VEL
LIN {X 0,Y 426.33,Z 333.519,A -85,B 0,C 180,E1 -18118.698,E2 -18118.698} C_VEL
LIN {X 0,Y 424.152,Z 324.536,A -85,B 0,C 180,E1 -18119.891,E2 -18119.891} C_VEL
LIN {X 0,Y 422.301,Z 318.332,A -85,B 0,C 180,E1 -18120.844,E2 -18120.844} C_VEL
LIN {X 0,Y 419.471,Z 313.383,A -85,B 0,C 180,E1 -18121.91,E2 -18121.91} C_VEL
LIN {X 0,Y 417.076,Z 309.229,A -85,B 0,C 180,E1 -18122.891,E2 -18122.891} C_VEL
LIN {X 0,Y 415.467,Z 306.365,A -85,B 0,C 180,E1 -18123.631,E2 -18123.631} C_VEL
LIN {X 0,Y 415.261,Z 305.318,A -85,B 0,C 180,E1 -18123.825,E2 -18123.825} C_VEL
LIN {X 0,Y 415.309,Z 305.312,A -85,B 0,C 180,E1 -18127.563,E2 -18127.563} C_VEL
LIN {X 0,Y 415.273,Z 305.313,A -85,B 0,C 180,E1 -18131.136,E2 -18131.136} C_VEL
LIN {X 0,Y 415.311,Z 305.307,A -85,B 0,C 180,E1 -18133.75,E2 -18133.75} C_VEL
LIN {X 0,Y 415.305,Z 305.309,A -85,B 0,C 180,E1 -18136.49,E2 -18136.49} C_VEL
LIN {X 0,Y 415.285,Z 305.312,A -85,B 0,C 180,E1 -18140.139,E2 -18140.139} C_VEL
LIN {X 0,Y 415.322,Z 305.309,A -85,B 0,C 180,E1 -18142.617,E2 -18142.617} C_VEL
LIN {X 0,Y 415.362,Z 305.302,A -85,B 0,C 180,E1 -18145.724,E2 -18145.724} C_VEL
LIN {X 0,Y 415.362,Z 305.305,A -85,B 0,C 180,E1 -18149.609,E2 -18149.609} C_VEL
LIN {X 0,Y 415.342,Z 305.307,A -85,B 0,C 180,E1 -18152.913,E2 -18152.913} C_VEL
LIN {X 0,Y 415.338,Z 305.322,A -85,B 0,C 180,E1 -18154.864,E2 -18154.864} C_VEL
LIN {X 0,Y 415.901,Z 307.286,A -85,B 0,C 180,E1 -18155.433,E2 -18155.433} C_VEL
LIN {X 0,Y 418.296,Z 312.506,A -85,B 0,C 180,E1 -18157.074,E2 -18157.074} C_VEL
LIN {X 0,Y 421.723,Z 321.706,A -85,B 0,C 180,E1 -18159.587,E2 -18159.587} C_VEL
LIN {X 0,Y 424.499,Z 330.402,A -85,B 0,C 180,E1 -18161.729,E2 -18161.729} C_VEL
LIN {X 0,Y 427.126,Z 340.861,A -85,B 0,C 180,E1 -18164.057,E2 -18164.057} C_VEL
LIN {X 0,Y 428.303,Z 346.942,A -85,B 0,C 180,E1 -18165.295,E2 -18165.295} C_VEL
LIN {X 0,Y 430.312,Z 351.999,A -85,B 0,C 180,E1 -18165.706,E2 -18165.706} C_VEL
LIN {X 0,Y 434.146,Z 368.505,A -85,B 0,C 180,E1 -18166.678,E2 -18166.678} C_VEL
LIN {X 0,Y 437.04,Z 385.299,A -85,B 0,C 180,E1 -18167.51,E2 -18167.51} C_VEL
LIN {X 0,Y 431.116,Z 487.701,A -85,B 0,C 180,E1 -18170,E2 -18170} C_VEL
LIN {X 0,Y 429.881,Z 502.763,A -85,B 0,C 180,E1 -18170.563,E2 -18170.563} C_VEL
LIN {X 0,Y 428.424,Z 517.058,A -85,B 0,C 180,E1 -18171.302,E2 -18171.302} C_VEL
LIN {X 0,Y 426.665,Z 530.898,A -85,B 0,C 180,E1 -18172.216,E2 -18172.216} C_VEL
LIN {X 0,Y 424.864,Z 543.316,A -85,B 0,C 180,E1 -18173.254,E2 -18173.254} C_VEL
LIN {X 0,Y 423.05,Z 554.872,A -85,B 0,C 180,E1 -18174.445,E2 -18174.445} C_VEL
LIN {X 0,Y 421.145,Z 566.364,A -85,B 0,C 180,E1 -18175.893,E2 -18175.893} C_VEL
LIN {X 0,Y 419.386,Z 575.967,A -85,B 0,C 180,E1 -18177.367,E2 -18177.367} C_VEL
LIN {X 0,Y 417.539,Z 584.822,A -85,B 0,C 180,E1 -18179.039,E2 -18179.039} C_VEL
LIN {X 0,Y 416.387,Z 591.046,A -85,B 0,C 180,E1 -18180.482,E2 -18180.482} C_VEL
LIN {X 0,Y 415.098,Z 597.632,A -85,B 0,C 180,E1 -18182.418,E2 -18182.418} C_VEL
LIN {X 0,Y 414.381,Z 602.171,A -85,B 0,C 180,E1 -18184.193,E2 -18184.193} C_VEL
LIN {X 0,Y 413.802,Z 605.216,A -85,B 0,C 180,E1 -18185.829,E2 -18185.829} C_VEL
LIN {X 0,Y 413.255,Z 607.487,A -85,B 0,C 180,E1 -18187.793,E2 -18187.793} C_VEL
LIN {X 0,Y 413.104,Z 608.309,A -85,B 0,C 180,E1 -18189.762,E2 -18189.762} C_VEL
LIN {X 0,Y 412.911,Z 607.675,A -85,B 0,C 180,E1 -18191.745,E2 -18191.745} C_VEL
LIN {X 0,Y 412.931,Z 605.495,A -85,B 0,C 180,E1 -18193.738,E2 -18193.738} C_VEL
LIN {X 0,Y 413.017,Z 603.64,A -85,B 0,C 180,E1 -18194.828,E2 -18194.828} C_VEL
LIN {X 0,Y 413.15,Z 599.192,A -85,B 0,C 180,E1 -18196.751,E2 -18196.751} C_VEL
LIN {X 0,Y 413.377,Z 594.081,A -85,B 0,C 180,E1 -18198.393,E2 -18198.393} C_VEL
LIN {X 0,Y 413.746,Z 587.576,A -85,B 0,C 180,E1 -18200.049,E2 -18200.049} C_VEL
LIN {X 0,Y 414.237,Z 578.775,A -85,B 0,C 180,E1 -18201.839,E2 -18201.839} C_VEL
LIN {X 0,Y 414.872,Z 569.416,A -85,B 0,C 180,E1 -18203.376,E2 -18203.376} C_VEL
LIN {X 0,Y 415.561,Z 559.167,A -85,B 0,C 180,E1 -18204.767,E2 -18204.767} C_VEL
LIN {X 0,Y 416.394,Z 547.554,A -85,B 0,C 180,E1 -18206.07,E2 -18206.07} C_VEL
LIN {X 0,Y 417.16,Z 536.03,A -85,B 0,C 180,E1 -18207.135,E2 -18207.135} C_VEL
LIN {X 0,Y 417.985,Z 522.901,A -85,B 0,C 180,E1 -18208.119,E2 -18208.119} C_VEL
LIN {X 0,Y 418.772,Z 508.809,A -85,B 0,C 180,E1 -18208.948,E2 -18208.948} C_VEL
LIN {X 0,Y 419.507,Z 494.095,A -85,B 0,C 180,E1 -18209.597,E2 -18209.597} C_VEL
LIN {X 0,Y 419.966,Z 480.303,A -85,B 0,C 180,E1 -18210.024,E2 -18210.024} C_VEL
LIN {X 0,Y 422.595,Z 376.989,A -85,B 0,C 180,E1 -18212.291,E2 -18212.291} C_VEL
LIN {X 0,Y 418.54,Z 344.426,A -85,B 0,C 180,E1 -18213.196,E2 -18213.196} C_VEL
LIN {X 0,Y 419.496,Z 326.234,A -85,B 0,C 180,E1 -18216.036,E2 -18216.036} C_VEL
LIN {X 0,Y 416.353,Z 310.319,A -85,B 0,C 180,E1 -18218.7,E2 -18218.7} C_VEL
LIN {X 0,Y 415.332,Z 305.307,A -85,B 0,C 180,E1 -18219.572,E2 -18219.572} C_VEL
LIN {X 0,Y 415.31,Z 305.306,A -85,B 0,C 180,E1 -18223.51,E2 -18223.51} C_VEL
LIN {X 0,Y 415.299,Z 305.313,A -85,B 0,C 180,E1 -18226.489,E2 -18226.489} C_VEL
LIN {X 0,Y 415.269,Z 305.316,A -85,B 0,C 180,E1 -18230.135,E2 -18230.135} C_VEL
LIN {X 0,Y 415.307,Z 305.309,A -85,B 0,C 180,E1 -18232.613,E2 -18232.613} C_VEL
LIN {X 0,Y 415.279,Z 305.314,A -85,B 0,C 180,E1 -18236.176,E2 -18236.176} C_VEL
LIN {X 0,Y 415.352,Z 305.302,A -85,B 0,C 180,E1 -18239.606,E2 -18239.606} C_VEL
LIN {X 0,Y 415.325,Z 305.303,A -85,B 0,C 180,E1 -18242.91,E2 -18242.91} C_VEL
LIN {X 0,Y 415.349,Z 305.308,A -85,B 0,C 180,E1 -18246.123,E2 -18246.123} C_VEL
LIN {X 0,Y 415.364,Z 305.3,A -85,B 0,C 180,E1 -18249.258,E2 -18249.258} C_VEL
LIN {X 0,Y 415.384,Z 305.299,A -85,B 0,C 180,E1 -18252.328,E2 -18252.328} C_VEL
LIN {X 0,Y 415.431,Z 305.293,A -85,B 0,C 180,E1 -18255.348,E2 -18255.348} C_VEL
LIN {X 0,Y 415.52,Z 305.283,A -85,B 0,C 180,E1 -18258.327,E2 -18258.327} C_VEL
LIN {X 0,Y 415.523,Z 305.486,A -85,B 0,C 180,E1 -18259.557,E2 -18259.557} C_VEL
LIN {X 0,Y 416.078,Z 308.436,A -85,B 0,C 180,E1 -18260.276,E2 -18260.276} C_VEL
LIN {X 0,Y 423.103,Z 329.953,A -85,B 0,C 180,E1 -18260.975,E2 -18260.975} C_VEL
LIN {X 0,Y 424.344,Z 337.247,A -85,B 0,C 180,E1 -18261.155,E2 -18261.155} C_VEL
LIN {X 0,Y 422.278,Z 444.348,A -85,B 0,C 180,E1 -18262.971,E2 -18262.971} C_VEL
LIN {X 0,Y 421.844,Z 458.693,A -85,B 0,C 180,E1 -18263.413,E2 -18263.413} C_VEL
LIN {X 0,Y 421.226,Z 472.48,A -85,B 0,C 180,E1 -18264.032,E2 -18264.032} C_VEL
LIN {X 0,Y 420.358,Z 486.229,A -85,B 0,C 180,E1 -18264.859,E2 -18264.859} C_VEL
LIN {X 0,Y 419.594,Z 497.13,A -85,B 0,C 180,E1 -18265.69,E2 -18265.69} C_VEL
LIN {X 0,Y 418.395,Z 508.724,A -85,B 0,C 180,E1 -18266.759,E2 -18266.759} C_VEL
LIN {X 0,Y 417.657,Z 518.298,A -85,B 0,C 180,E1 -18267.835,E2 -18267.835} C_VEL
LIN {X 0,Y 416.79,Z 527.337,A -85,B 0,C 180,E1 -18269.035,E2 -18269.035} C_VEL
LIN {X 0,Y 415.818,Z 536.428,A -85,B 0,C 180,E1 -18270.48,E2 -18270.48} C_VEL
LIN {X 0,Y 415.113,Z 543.993,A -85,B 0,C 180,E1 -18271.932,E2 -18271.932} C_VEL
LIN {X 0,Y 414.61,Z 550.299,A -85,B 0,C 180,E1 -18273.387,E2 -18273.387} C_VEL
LIN {X 0,Y 414.271,Z 555.477,A -85,B 0,C 180,E1 -18274.847,E2 -18274.847} C_VEL
LIN {X 0,Y 413.778,Z 560.979,A -85,B 0,C 180,E1 -18276.803,E2 -18276.803} C_VEL
LIN {X 0,Y 413.456,Z 564.912,A -85,B 0,C 180,E1 -18278.768,E2 -18278.768} C_VEL
LIN {X 0,Y 413.411,Z 567.408,A -85,B 0,C 180,E1 -18280.739,E2 -18280.739} C_VEL
LIN {X 0,Y 413.398,Z 568.558,A -85,B 0,C 180,E1 -18282.722,E2 -18282.722} C_VEL
LIN {X 0,Y 413.637,Z 568.352,A -85,B 0,C 180,E1 -18284.712,E2 -18284.712} C_VEL
LIN {X 0,Y 413.963,Z 566.782,A -85,B 0,C 180,E1 -18286.714,E2 -18286.714} C_VEL
LIN {X 0,Y 414.604,Z 563.787,A -85,B 0,C 180,E1 -18288.72,E2 -18288.72} C_VEL
LIN {X 0,Y 415.508,Z 559.265,A -85,B 0,C 180,E1 -18290.73,E2 -18290.73} C_VEL
LIN {X 0,Y 416.379,Z 554.529,A -85,B 0,C 180,E1 -18292.298,E2 -18292.298} C_VEL
LIN {X 0,Y 417.598,Z 548.095,A -85,B 0,C 180,E1 -18293.998,E2 -18293.998} C_VEL
LIN {X 0,Y 419.199,Z 539.779,A -85,B 0,C 180,E1 -18295.746,E2 -18295.746} C_VEL
LIN {X 0,Y 420.186,Z 533.847,A -85,B 0,C 180,E1 -18296.785,E2 -18296.785} C_VEL
LIN {X 0,Y 420.224,Z 530.136,A -85,B 0,C 180,E1 -18297.41,E2 -18297.41} C_VEL
LIN {X 0,Y 418.657,Z 523.958,A -85,B 0,C 180,E1 -18298.449,E2 -18298.449} C_VEL
LIN {X 0,Y 417.07,Z 517.372,A -85,B 0,C 180,E1 -18299.44,E2 -18299.44} C_VEL
LIN {X 0,Y 417.066,Z 512.98,A -85,B 0,C 180,E1 -18299.982,E2 -18299.982} C_VEL
LIN {X 0,Y 418.667,Z 501.771,A -85,B 0,C 180,E1 -18301.098,E2 -18301.098} C_VEL
LIN {X 0,Y 420.221,Z 489.006,A -85,B 0,C 180,E1 -18302.121,E2 -18302.121} C_VEL
LIN {X 0,Y 421.482,Z 475.476,A -85,B 0,C 180,E1 -18302.971,E2 -18302.971} C_VEL
LIN {X 0,Y 422.453,Z 462.385,A -85,B 0,C 180,E1 -18303.592,E2 -18303.592} C_VEL
LIN {X 0,Y 423.18,Z 448.553,A -85,B 0,C 180,E1 -18304.055,E2 -18304.055} C_VEL
LIN {X 0,Y 423.622,Z 428.904,A -85,B 0,C 180,E1 -18304.454,E2 -18304.454} C_VEL
LIN {X 0,Y 425.802,Z 346.562,A -85,B 0,C 180,E1 -18305.851,E2 -18305.851} C_VEL
LIN {X 0,Y 416.741,Z 325.854,A -85,B 0,C 180,E1 -18306.926,E2 -18306.926} C_VEL
LIN {X 0,Y 409.222,Z 310.313,A -85,B 0,C 180,E1 -18307.861,E2 -18307.861} C_VEL
LIN {X 0,Y 408.215,Z 306.188,A -85,B 0,C 180,E1 -18309.089,E2 -18309.089} C_VEL
LIN {X 0,Y 408.219,Z 306.19,A -85,B 0,C 180,E1 -18312.454,E2 -18312.454} C_VEL
LIN {X 0,Y 408.255,Z 306.173,A -85,B 0,C 180,E1 -18315.296,E2 -18315.296} C_VEL
LIN {X 0,Y 408.234,Z 306.191,A -85,B 0,C 180,E1 -18319.016,E2 -18319.016} C_VEL
LIN {X 0,Y 408.253,Z 306.187,A -85,B 0,C 180,E1 -18322.108,E2 -18322.108} C_VEL
LIN {X 0,Y 408.283,Z 306.165,A -85,B 0,C 180,E1 -18325.518,E2 -18325.518} C_VEL
LIN {X 0,Y 408.277,Z 306.178,A -85,B 0,C 180,E1 -18329.065,E2 -18329.065} C_VEL
LIN {X 0,Y 408.278,Z 306.175,A -85,B 0,C 180,E1 -18332.405,E2 -18332.405} C_VEL
LIN {X 0,Y 408.295,Z 306.178,A -85,B 0,C 180,E1 -18335.687,E2 -18335.687} C_VEL
LIN {X 0,Y 408.287,Z 306.184,A -85,B 0,C 180,E1 -18338.883,E2 -18338.883} C_VEL
LIN {X 0,Y 408.358,Z 306.165,A -85,B 0,C 180,E1 -18340.98,E2 -18340.98} C_VEL
LIN {X 0,Y 408.341,Z 306.175,A -85,B 0,C 180,E1 -18344.07,E2 -18344.07} C_VEL
LIN {X 0,Y 408.464,Z 306.163,A -85,B 0,C 180,E1 -18347.794,E2 -18347.794} C_VEL
LIN {X 0,Y 408.458,Z 306.149,A -85,B 0,C 180,E1 -18351.122,E2 -18351.122} C_VEL
LIN {X 0,Y 408.578,Z 306.146,A -85,B 0,C 180,E1 -18354.096,E2 -18354.096} C_VEL
LIN {X 0,Y 408.582,Z 306.134,A -85,B 0,C 180,E1 -18357.052,E2 -18357.052} C_VEL
LIN {X 0,Y 408.574,Z 306.145,A -85,B 0,C 180,E1 -18360,E2 -18360} C_VEL
LIN {X 0,Y 408.591,Z 306.143,A -85,B 0,C 180,E1 -18363.932,E2 -18363.932} C_VEL
LIN {X 0,Y 408.53,Z 306.139,A -85,B 0,C 180,E1 -18366.893,E2 -18366.893} C_VEL
LIN {X 0,Y 408.468,Z 306.158,A -85,B 0,C 180,E1 -18369.874,E2 -18369.874} C_VEL
LIN {X 0,Y 408.415,Z 306.153,A -85,B 0,C 180,E1 -18372.883,E2 -18372.883} C_VEL
LIN {X 0,Y 408.388,Z 306.167,A -85,B 0,C 180,E1 -18376.174,E2 -18376.174} C_VEL
LIN {X 0,Y 408.363,Z 306.172,A -85,B 0,C 180,E1 -18379.381,E2 -18379.381} C_VEL
LIN {X 0,Y 408.281,Z 306.181,A -85,B 0,C 180,E1 -18383.24,E2 -18383.24} C_VEL
LIN {X 0,Y 408.285,Z 306.177,A -85,B 0,C 180,E1 -18386.869,E2 -18386.869} C_VEL
LIN {X 0,Y 408.277,Z 306.182,A -85,B 0,C 180,E1 -18389.837,E2 -18389.837} C_VEL
LIN {X 0,Y 408.269,Z 306.182,A -85,B 0,C 180,E1 -18393.299,E2 -18393.299} C_VEL
LIN {X 0,Y 408.332,Z 306.146,A -85,B 0,C 180,E1 -18396.276,E2 -18396.276} C_VEL
LIN {X 0,Y 408.324,Z 306.178,A -85,B 0,C 180,E1 -18399.477,E2 -18399.477} C_VEL
LIN {X 0,Y 408.28,Z 306.182,A -85,B 0,C 180,E1 -18403.333,E2 -18403.333} C_VEL
LIN {X 0,Y 408.284,Z 306.184,A -85,B 0,C 180,E1 -18406.672,E2 -18406.672} C_VEL
LIN {X 0,Y 408.327,Z 306.181,A -85,B 0,C 180,E1 -18410.528,E2 -18410.528} C_VEL
LIN {X 0,Y 408.337,Z 306.171,A -85,B 0,C 180,E1 -18413.728,E2 -18413.728} C_VEL
LIN {X 0,Y 408.346,Z 306.275,A -85,B 0,C 180,E1 -18414.762,E2 -18414.762} C_VEL
LIN {X 0,Y 411.659,Z 319.191,A -85,B 0,C 180,E1 -18417.881,E2 -18417.881} C_VEL
LIN {X 0,Y 414.623,Z 332.416,A -85,B 0,C 180,E1 -18420.879,E2 -18420.879} C_VEL
LIN {X 0,Y 416.287,Z 340.904,A -85,B 0,C 180,E1 -18422.712,E2 -18422.712} C_VEL
LIN {X 0,Y 415.905,Z 345.341,A -85,B 0,C 180,E1 -18423.562,E2 -18423.562} C_VEL
LIN {X 0,Y 414.986,Z 351.357,A -85,B 0,C 180,E1 -18424.681,E2 -18424.681} C_VEL
LIN {X 0,Y 420.88,Z 382.303,A -85,B 0,C 180,E1 -18425.718,E2 -18425.718} C_VEL
LIN {X 0,Y 424.355,Z 405.59,A -85,B 0,C 180,E1 -18426.405,E2 -18426.405} C_VEL
LIN {X 0,Y 422.858,Z 467.888,A -85,B 0,C 180,E1 -18427.471,E2 -18427.471} C_VEL
LIN {X 0,Y 422.21,Z 491.967,A -85,B 0,C 180,E1 -18427.925,E2 -18427.925} C_VEL
LIN {X 0,Y 421.146,Z 506.554,A -85,B 0,C 180,E1 -18428.38,E2 -18428.38} C_VEL
LIN {X 0,Y 419.76,Z 519.915,A -85,B 0,C 180,E1 -18428.978,E2 -18428.978} C_VEL
LIN {X 0,Y 418.281,Z 532.57,A -85,B 0,C 180,E1 -18429.738,E2 -18429.738} C_VEL
LIN {X 0,Y 416.501,Z 545.563,A -85,B 0,C 180,E1 -18430.732,E2 -18430.732} C_VEL
LIN {X 0,Y 414.545,Z 557.9,A -85,B 0,C 180,E1 -18431.915,E2 -18431.915} C_VEL
LIN {X 0,Y 412.569,Z 568.959,A -85,B 0,C 180,E1 -18433.227,E2 -18433.227} C_VEL
LIN {X 0,Y 410.869,Z 578.933,A -85,B 0,C 180,E1 -18434.681,E2 -18434.681} C_VEL
LIN {X 0,Y 409.489,Z 587.252,A -85,B 0,C 180,E1 -18436.147,E2 -18436.147} C_VEL
LIN {X 0,Y 408.353,Z 594.433,A -85,B 0,C 180,E1 -18437.672,E2 -18437.672} C_VEL
LIN {X 0,Y 407.205,Z 601.712,A -85,B 0,C 180,E1 -18439.597,E2 -18439.597} C_VEL
LIN {X 0,Y 406.459,Z 607.494,A -85,B 0,C 180,E1 -18441.58,E2 -18441.58} C_VEL
LIN {X 0,Y 406.224,Z 610.833,A -85,B 0,C 180,E1 -18443.07,E2 -18443.07} C_VEL
LIN {X 0,Y 406.163,Z 613.558,A -85,B 0,C 180,E1 -18444.56,E2 -18444.56} C_VEL
LIN {X 0,Y 406.091,Z 617.576,A -85,B 0,C 180,E1 -18446.046,E2 -18446.046} C_VEL
LIN {X 0,Y 406.104,Z 619.697,A -85,B 0,C 180,E1 -18447.036,E2 -18447.036} C_VEL
LIN {X 0,Y 406.124,Z 622.76,A -85,B 0,C 180,E1 -18449.014,E2 -18449.014} C_VEL
LIN {X 0,Y 406.08,Z 624.32,A -85,B 0,C 180,E1 -18450.991,E2 -18450.991} C_VEL
LIN {X 0,Y 405.994,Z 624.417,A -85,B 0,C 180,E1 -18452.969,E2 -18452.969} C_VEL
LIN {X 0,Y 406.11,Z 623.077,A -85,B 0,C 180,E1 -18454.95,E2 -18454.95} C_VEL
LIN {X 0,Y 406.396,Z 620.262,A -85,B 0,C 180,E1 -18456.932,E2 -18456.932} C_VEL
LIN {X 0,Y 406.939,Z 615.93,A -85,B 0,C 180,E1 -18458.914,E2 -18458.914} C_VEL
LIN {X 0,Y 408.126,Z 609.975,A -85,B 0,C 180,E1 -18460.884,E2 -18460.884} C_VEL
LIN {X 0,Y 409.275,Z 602.887,A -85,B 0,C 180,E1 -18462.705,E2 -18462.705} C_VEL
LIN {X 0,Y 410.781,Z 595.04,A -85,B 0,C 180,E1 -18464.317,E2 -18464.317} C_VEL
LIN {X 0,Y 412.456,Z 586.417,A -85,B 0,C 180,E1 -18465.769,E2 -18465.769} C_VEL
LIN {X 0,Y 414.221,Z 576.089,A -85,B 0,C 180,E1 -18467.215,E2 -18467.215} C_VEL
LIN {X 0,Y 416.088,Z 565.781,A -85,B 0,C 180,E1 -18468.402,E2 -18468.402} C_VEL
LIN {X 0,Y 418.043,Z 553.374,A -85,B 0,C 180,E1 -18469.581,E2 -18469.581} C_VEL
LIN {X 0,Y 420.067,Z 539.939,A -85,B 0,C 180,E1 -18470.606,E2 -18470.606} C_VEL
LIN {X 0,Y 421.804,Z 526.223,A -85,B 0,C 180,E1 -18471.43,E2 -18471.43} C_VEL
LIN {X 0,Y 423.458,Z 510.912,A -85,B 0,C 180,E1 -18472.107,E2 -18472.107} C_VEL
LIN {X 0,Y 424.743,Z 495.525,A -85,B 0,C 180,E1 -18472.579,E2 -18472.579} C_VEL
LIN {X 0,Y 429.885,Z 407.071,A -85,B 0,C 180,E1 -18474.794,E2 -18474.794} C_VEL
LIN {X 0,Y 428.708,Z 391.485,A -85,B 0,C 180,E1 -18475.423,E2 -18475.423} C_VEL
LIN {X 0,Y 426.424,Z 372.162,A -85,B 0,C 180,E1 -18476.33,E2 -18476.33} C_VEL
LIN {X 0,Y 423.293,Z 353.409,A -85,B 0,C 180,E1 -18477.378,E2 -18477.378} C_VEL
LIN {X 0,Y 422.907,Z 345.261,A -85,B 0,C 180,E1 -18478.121,E2 -18478.121} C_VEL
LIN {X 0,Y 421.216,Z 337.704,A -85,B 0,C 180,E1 -18479.043,E2 -18479.043} C_VEL
LIN {X 0,Y 419.016,Z 328.445,A -85,B 0,C 180,E1 -18480.299,E2 -18480.299} C_VEL
LIN {X 0,Y 417.437,Z 323.047,A -85,B 0,C 180,E1 -18481.156,E2 -18481.156} C_VEL
LIN {X 0,Y 413.29,Z 315.47,A -85,B 0,C 180,E1 -18482.845,E2 -18482.845} C_VEL
LIN {X 0,Y 409.069,Z 308.744,A -85,B 0,C 180,E1 -18484.725,E2 -18484.725} C_VEL
LIN {X 0,Y 408.224,Z 306.193,A -85,B 0,C 180,E1 -18485.389,E2 -18485.389} C_VEL
LIN {X 0,Y 408.255,Z 306.188,A -85,B 0,C 180,E1 -18488.147,E2 -18488.147} C_VEL
LIN {X 0,Y 408.242,Z 306.188,A -85,B 0,C 180,E1 -18492.004,E2 -18492.004} C_VEL
LIN {X 0,Y 408.277,Z 306.183,A -85,B 0,C 180,E1 -18495.299,E2 -18495.299} C_VEL
LIN {X 0,Y 408.242,Z 306.192,A -85,B 0,C 180,E1 -18499.022,E2 -18499.022} C_VEL
LIN {X 0,Y 408.271,Z 306.188,A -85,B 0,C 180,E1 -18502.113,E2 -18502.113} C_VEL
LIN {X 0,Y 408.31,Z 306.182,A -85,B 0,C 180,E1 -18505.521,E2 -18505.521} C_VEL
LIN {X 0,Y 408.304,Z 306.183,A -85,B 0,C 180,E1 -18509.068,E2 -18509.068} C_VEL
LIN {X 0,Y 408.305,Z 306.184,A -85,B 0,C 180,E1 -18512.407,E2 -18512.407} C_VEL
LIN {X 0,Y 408.349,Z 306.263,A -85,B 0,C 180,E1 -18513.444,E2 -18513.444} C_VEL
LIN {X 0,Y 408.92,Z 308.333,A -85,B 0,C 180,E1 -18514.1,E2 -18514.1} C_VEL
LIN {X 0,Y 410.055,Z 310.393,A -85,B 0,C 180,E1 -18514.871,E2 -18514.871} C_VEL
LIN {X 0,Y 413.243,Z 318.202,A -85,B 0,C 180,E1 -18517.332,E2 -18517.332} C_VEL
LIN {X 0,Y 416.117,Z 326.184,A -85,B 0,C 180,E1 -18519.557,E2 -18519.557} C_VEL
LIN {X 0,Y 418.793,Z 334.829,A -85,B 0,C 180,E1 -18521.724,E2 -18521.724} C_VEL
LIN {X 0,Y 421.047,Z 344.181,A -85,B 0,C 180,E1 -18523.845,E2 -18523.845} C_VEL
LIN {X 0,Y 421.661,Z 347.242,A -85,B 0,C 180,E1 -18524.471,E2 -18524.471} C_VEL
LIN {X 0,Y 425.125,Z 354.965,A -85,B 0,C 180,E1 -18525.187,E2 -18525.187} C_VEL
LIN {X 0,Y 428.633,Z 370.362,A -85,B 0,C 180,E1 -18526.125,E2 -18526.125} C_VEL
LIN {X 0,Y 431.375,Z 386.684,A -85,B 0,C 180,E1 -18526.964,E2 -18526.964} C_VEL
LIN {X 0,Y 425.145,Z 488.464,A -85,B 0,C 180,E1 -18529.499,E2 -18529.499} C_VEL
LIN {X 0,Y 423.848,Z 503.231,A -85,B 0,C 180,E1 -18530.067,E2 -18530.067} C_VEL
LIN {X 0,Y 422.319,Z 517.453,A -85,B 0,C 180,E1 -18530.814,E2 -18530.814} C_VEL
LIN {X 0,Y 420.47,Z 531.218,A -85,B 0,C 180,E1 -18531.739,E2 -18531.739} C_VEL
LIN {X 0,Y 418.588,Z 543.561,A -85,B 0,C 180,E1 -18532.79,E2 -18532.79} C_VEL
LIN {X 0,Y 416.539,Z 555.893,A -85,B 0,C 180,E1 -18534.088,E2 -18534.088} C_VEL
LIN {X 0,Y 414.715,Z 566.27,A -85,B 0,C 180,E1 -18535.422,E2 -18535.422} C_VEL
LIN {X 0,Y 412.95,Z 575.419,A -85,B 0,C 180,E1 -18536.84,E2 -18536.84} C_VEL
LIN {X 0,Y 410.98,Z 584.457,A -85,B 0,C 180,E1 -18538.535,E2 -18538.535} C_VEL
LIN {X 0,Y 409.703,Z 590.746,A -85,B 0,C 180,E1 -18540,E2 -18540} C_VEL
LIN {X 0,Y 408.618,Z 595.931,A -85,B 0,C 180,E1 -18541.473,E2 -18541.473} C_VEL
LIN {X 0,Y 407.535,Z 601.387,A -85,B 0,C 180,E1 -18543.449,E2 -18543.449} C_VEL
LIN {X 0,Y 407.014,Z 604.519,A -85,B 0,C 180,E1 -18545.034,E2 -18545.034} C_VEL
LIN {X 0,Y 406.386,Z 607.116,A -85,B 0,C 180,E1 -18546.93,E2 -18546.93} C_VEL
LIN {X 0,Y 406.067,Z 608.397,A -85,B 0,C 180,E1 -18548.931,E2 -18548.931} C_VEL
LIN {X 0,Y 405.953,Z 608.374,A -85,B 0,C 180,E1 -18550.416,E2 -18550.416} C_VEL
LIN {X 0,Y 405.803,Z 607.53,A -85,B 0,C 180,E1 -18551.954,E2 -18551.954} C_VEL
LIN {X 0,Y 405.844,Z 605.074,A -85,B 0,C 180,E1 -18553.982,E2 -18553.982} C_VEL
LIN {X 0,Y 405.944,Z 602.182,A -85,B 0,C 180,E1 -18555.512,E2 -18555.512} C_VEL
LIN {X 0,Y 406.089,Z 598.324,A -85,B 0,C 180,E1 -18557.051,E2 -18557.051} C_VEL
LIN {X 0,Y 406.368,Z 592.782,A -85,B 0,C 180,E1 -18558.759,E2 -18558.759} C_VEL
LIN {X 0,Y 406.753,Z 586.061,A -85,B 0,C 180,E1 -18560.409,E2 -18560.409} C_VEL
LIN {X 0,Y 407.167,Z 578.606,A -85,B 0,C 180,E1 -18561.909,E2 -18561.909} C_VEL
LIN {X 0,Y 407.843,Z 568.759,A -85,B 0,C 180,E1 -18563.535,E2 -18563.535} C_VEL
LIN {X 0,Y 408.51,Z 558.69,A -85,B 0,C 180,E1 -18564.907,E2 -18564.907} C_VEL
LIN {X 0,Y 409.42,Z 546.524,A -85,B 0,C 180,E1 -18566.275,E2 -18566.275} C_VEL
LIN {X 0,Y 410.269,Z 533.561,A -85,B 0,C 180,E1 -18567.449,E2 -18567.449} C_VEL
LIN {X 0,Y 411.091,Z 520.165,A -85,B 0,C 180,E1 -18568.426,E2 -18568.426} C_VEL
LIN {X 0,Y 411.89,Z 506.635,A -85,B 0,C 180,E1 -18569.199,E2 -18569.199} C_VEL
LIN {X 0,Y 412.567,Z 492.456,A -85,B 0,C 180,E1 -18569.808,E2 -18569.808} C_VEL
LIN {X 0,Y 413.051,Z 477.563,A -85,B 0,C 180,E1 -18570.245,E2 -18570.245} C_VEL
LIN {X 0,Y 415.649,Z 377.346,A -85,B 0,C 180,E1 -18572.498,E2 -18572.498} C_VEL
LIN {X 0,Y 411.596,Z 344.578,A -85,B 0,C 180,E1 -18573.422,E2 -18573.422} C_VEL
LIN {X 0,Y 412.514,Z 329.09,A -85,B 0,C 180,E1 -18575.859,E2 -18575.859} C_VEL
LIN {X 0,Y 411.964,Z 324.283,A -85,B 0,C 180,E1 -18576.649,E2 -18576.649} C_VEL
LIN {X 0,Y 408.311,Z 306.182,A -85,B 0,C 180,E1 -18579.732,E2 -18579.732} C_VEL
LIN {X 0,Y 408.252,Z 306.186,A -85,B 0,C 180,E1 -18583.337,E2 -18583.337} C_VEL
LIN {X 0,Y 408.241,Z 306.19,A -85,B 0,C 180,E1 -18586.659,E2 -18586.659} C_VEL
LIN {X 0,Y 408.222,Z 306.188,A -85,B 0,C 180,E1 -18589.304,E2 -18589.304} C_VEL
LIN {X 0,Y 408.261,Z 306.189,A -85,B 0,C 180,E1 -18592.112,E2 -18592.112} C_VEL
LIN {X 0,Y 408.263,Z 306.182,A -85,B 0,C 180,E1 -18595.514,E2 -18595.514} C_VEL
LIN {X 0,Y 408.268,Z 306.183,A -85,B 0,C 180,E1 -18599.073,E2 -18599.073} C_VEL
LIN {X 0,Y 408.285,Z 306.184,A -85,B 0,C 180,E1 -18602.404,E2 -18602.404} C_VEL
LIN {X 0,Y 408.307,Z 306.181,A -85,B 0,C 180,E1 -18605.685,E2 -18605.685} C_VEL
LIN {X 0,Y 408.314,Z 306.178,A -85,B 0,C 180,E1 -18608.883,E2 -18608.883} C_VEL
LIN {X 0,Y 408.388,Z 306.168,A -85,B 0,C 180,E1 -18610.979,E2 -18610.979} C_VEL
LIN {X 0,Y 408.408,Z 306.172,A -85,B 0,C 180,E1 -18614.071,E2 -18614.071} C_VEL
LIN {X 0,Y 408.491,Z 306.162,A -85,B 0,C 180,E1 -18617.792,E2 -18617.792} C_VEL
LIN {X 0,Y 408.44,Z 306.242,A -85,B 0,C 180,E1 -18619.312,E2 -18619.312} C_VEL
LIN {X 0,Y 408.958,Z 308.877,A -85,B 0,C 180,E1 -18619.961,E2 -18619.961} C_VEL
LIN {X 0,Y 416.543,Z 331.948,A -85,B 0,C 180,E1 -18620.724,E2 -18620.724} C_VEL
LIN {X 0,Y 417.583,Z 337.41,A -85,B 0,C 180,E1 -18620.868,E2 -18620.868} C_VEL
LIN {X 0,Y 415.464,Z 444.299,A -85,B 0,C 180,E1 -18622.703,E2 -18622.703} C_VEL
LIN {X 0,Y 415.009,Z 458.805,A -85,B 0,C 180,E1 -18623.152,E2 -18623.152} C_VEL
LIN {X 0,Y 414.416,Z 472.105,A -85,B 0,C 180,E1 -18623.751,E2 -18623.751} C_VEL
LIN {X 0,Y 413.571,Z 485.154,A -85,B 0,C 180,E1 -18624.531,E2 -18624.531} C_VEL
LIN {X 0,Y 412.644,Z 497.759,A -85,B 0,C 180,E1 -18625.495,E2 -18625.495} C_VEL
LIN {X 0,Y 411.435,Z 509.31,A -85,B 0,C 180,E1 -18626.582,E2 -18626.582} C_VEL
LIN {X 0,Y 410.627,Z 519.813,A -85,B 0,C 180,E1 -18627.798,E2 -18627.798} C_VEL
LIN {X 0,Y 409.499,Z 530.303,A -85,B 0,C 180,E1 -18629.263,E2 -18629.263} C_VEL
LIN {X 0,Y 408.65,Z 538.95,A -85,B 0,C 180,E1 -18630.734,E2 -18630.734} C_VEL
LIN {X 0,Y 407.822,Z 546.167,A -85,B 0,C 180,E1 -18632.212,E2 -18632.212} C_VEL
LIN {X 0,Y 407.426,Z 553.038,A -85,B 0,C 180,E1 -18633.941,E2 -18633.941} C_VEL
LIN {X 0,Y 407.011,Z 557.826,A -85,B 0,C 180,E1 -18635.429,E2 -18635.429} C_VEL
LIN {X 0,Y 406.564,Z 562.795,A -85,B 0,C 180,E1 -18637.422,E2 -18637.422} C_VEL
LIN {X 0,Y 406.364,Z 565.537,A -85,B 0,C 180,E1 -18638.922,E2 -18638.922} C_VEL
LIN {X 0,Y 406.301,Z 567.943,A -85,B 0,C 180,E1 -18640.929,E2 -18640.929} C_VEL
LIN {X 0,Y 406.339,Z 569,A -85,B 0,C 180,E1 -18642.947,E2 -18642.947} C_VEL
LIN {X 0,Y 406.616,Z 568.702,A -85,B 0,C 180,E1 -18644.972,E2 -18644.972} C_VEL
LIN {X 0,Y 406.963,Z 567.04,A -85,B 0,C 180,E1 -18647.011,E2 -18647.011} C_VEL
LIN {X 0,Y 407.693,Z 563.855,A -85,B 0,C 180,E1 -18649.102,E2 -18649.102} C_VEL
LIN {X 0,Y 408.628,Z 559.279,A -85,B 0,C 180,E1 -18651.095,E2 -18651.095} C_VEL
LIN {X 0,Y 409.61,Z 554.369,A -85,B 0,C 180,E1 -18652.719,E2 -18652.719} C_VEL
LIN {X 0,Y 410.895,Z 547.914,A -85,B 0,C 180,E1 -18654.415,E2 -18654.415} C_VEL
LIN {X 0,Y 412.552,Z 539.396,A -85,B 0,C 180,E1 -18656.192,E2 -18656.192} C_VEL
LIN {X 0,Y 414.172,Z 530.425,A -85,B 0,C 180,E1 -18657.712,E2 -18657.712} C_VEL
LIN {X 0,Y 415.827,Z 520.712,A -85,B 0,C 180,E1 -18659.067,E2 -18659.067} C_VEL
LIN {X 0,Y 417.066,Z 512.98,A -85,B 0,C 180,E1 -18659.982,E2 -18659.982} C_VEL
LIN {X 0,Y 417.064,Z 508.444,A -85,B 0,C 180,E1 -18660.505,E2 -18660.505} C_VEL
LIN {X 0,Y 415.492,Z 501.017,A -85,B 0,C 180,E1 -18661.386,E2 -18661.386} C_VEL
LIN {X 0,Y 413.92,Z 493.23,A -85,B 0,C 180,E1 -18662.2,E2 -18662.2} C_VEL
LIN {X 0,Y 413.896,Z 488.141,A -85,B 0,C 180,E1 -18662.611,E2 -18662.611} C_VEL
LIN {X 0,Y 415.19,Z 474.428,A -85,B 0,C 180,E1 -18663.463,E2 -18663.463} C_VEL
LIN {X 0,Y 416.24,Z 460.724,A -85,B 0,C 180,E1 -18664.094,E2 -18664.094} C_VEL
LIN {X 0,Y 416.913,Z 446.95,A -85,B 0,C 180,E1 -18664.537,E2 -18664.537} C_VEL
LIN {X 0,Y 417.82,Z 410.812,A -85,B 0,C 180,E1 -18665.204,E2 -18665.204} C_VEL
LIN {X 0,Y 419.533,Z 348.492,A -85,B 0,C 180,E1 -18666.275,E2 -18666.275} C_VEL
LIN {X 0,Y 411.113,Z 329.223,A -85,B 0,C 180,E1 -18667.302,E2 -18667.302} C_VEL
LIN {X 0,Y 402.113,Z 310.85,A -85,B 0,C 180,E1 -18668.435,E2 -18668.435} C_VEL
LIN {X 0,Y 401.182,Z 307.068,A -85,B 0,C 180,E1 -18669.567,E2 -18669.567} C_VEL
LIN {X 0,Y 401.18,Z 307.073,A -85,B 0,C 180,E1 -18672.912,E2 -18672.912} C_VEL
LIN {X 0,Y 401.227,Z 307.052,A -85,B 0,C 180,E1 -18675.709,E2 -18675.709} C_VEL
LIN {X 0,Y 401.179,Z 307.071,A -85,B 0,C 180,E1 -18678.652,E2 -18678.652} C_VEL
LIN {X 0,Y 401.211,Z 307.061,A -85,B 0,C 180,E1 -18682.335,E2 -18682.335} C_VEL
LIN {X 0,Y 401.224,Z 307.052,A -85,B 0,C 180,E1 -18686.038,E2 -18686.038} C_VEL
LIN {X 0,Y 401.223,Z 307.058,A -85,B 0,C 180,E1 -18689.584,E2 -18689.584} C_VEL
LIN {X 0,Y 401.242,Z 307.051,A -85,B 0,C 180,E1 -18693.007,E2 -18693.007} C_VEL
LIN {X 0,Y 401.246,Z 307.05,A -85,B 0,C 180,E1 -18696.328,E2 -18696.328} C_VEL
LIN {X 0,Y 401.249,Z 307.059,A -85,B 0,C 180,E1 -18699.566,E2 -18699.566} C_VEL
LIN {X 0,Y 401.264,Z 307.05,A -85,B 0,C 180,E1 -18701.687,E2 -18701.687} C_VEL
LIN {X 0,Y 401.279,Z 307.053,A -85,B 0,C 180,E1 -18704.821,E2 -18704.821} C_VEL
LIN {X 0,Y 401.414,Z 307.041,A -85,B 0,C 180,E1 -18707.913,E2 -18707.913} C_VEL
LIN {X 0,Y 401.46,Z 307.027,A -85,B 0,C 180,E1 -18711.977,E2 -18711.977} C_VEL
LIN {X 0,Y 401.559,Z 307.017,A -85,B 0,C 180,E1 -18714.997,E2 -18714.997} C_VEL
LIN {X 0,Y 401.446,Z 307.033,A -85,B 0,C 180,E1 -18718,E2 -18718} C_VEL
LIN {X 0,Y 401.462,Z 307.022,A -85,B 0,C 180,E1 -18721,E2 -18721} C_VEL
LIN {X 0,Y 401.56,Z 307.019,A -85,B 0,C 180,E1 -18724.001,E2 -18724.001} C_VEL
LIN {X 0,Y 401.481,Z 307.016,A -85,B 0,C 180,E1 -18727.015,E2 -18727.015} C_VEL
LIN {X 0,Y 401.412,Z 307.037,A -85,B 0,C 180,E1 -18730.049,E2 -18730.049} C_VEL
LIN {X 0,Y 401.357,Z 307.033,A -85,B 0,C 180,E1 -18733.113,E2 -18733.113} C_VEL
LIN {X 0,Y 401.336,Z 307.044,A -85,B 0,C 180,E1 -18736.292,E2 -18736.292} C_VEL
LIN {X 0,Y 401.299,Z 307.051,A -85,B 0,C 180,E1 -18739.528,E2 -18739.528} C_VEL
LIN {X 0,Y 401.25,Z 307.049,A -85,B 0,C 180,E1 -18742.584,E2 -18742.584} C_VEL
LIN {X 0,Y 401.262,Z 307.053,A -85,B 0,C 180,E1 -18745.875,E2 -18745.875} C_VEL
LIN {X 0,Y 401.249,Z 307.058,A -85,B 0,C 180,E1 -18749.261,E2 -18749.261} C_VEL
LIN {X 0,Y 401.24,Z 307.061,A -85,B 0,C 180,E1 -18752.763,E2 -18752.763} C_VEL
LIN {X 0,Y 401.298,Z 307.023,A -85,B 0,C 180,E1 -18756.402,E2 -18756.402} C_VEL
LIN {X 0,Y 401.265,Z 307.059,A -85,B 0,C 180,E1 -18758.933,E2 -18758.933} C_VEL
LIN {X 0,Y 401.217,Z 307.061,A -85,B 0,C 180,E1 -18762.911,E2 -18762.911} C_VEL
LIN {X 0,Y 401.263,Z 307.056,A -85,B 0,C 180,E1 -18765.718,E2 -18765.718} C_VEL
LIN {X 0,Y 401.24,Z 307.063,A -85,B 0,C 180,E1 -18768.647,E2 -18768.647} C_VEL
LIN {X 0,Y 401.285,Z 307.059,A -85,B 0,C 180,E1 -18772.347,E2 -18772.347} C_VEL
LIN {X 0,Y 401.305,Z 307.105,A -85,B 0,C 180,E1 -18774.221,E2 -18774.221} C_VEL
LIN {X 0,Y 404.787,Z 320.543,A -85,B 0,C 180,E1 -18777.563,E2 -18777.563} C_VEL
LIN {X 0,Y 407.789,Z 334.126,A -85,B 0,C 180,E1 -18780.687,E2 -18780.687} C_VEL
LIN {X 0,Y 409.412,Z 342.291,A -85,B 0,C 180,E1 -18782.491,E2 -18782.491} C_VEL
LIN {X 0,Y 409.536,Z 343.741,A -85,B 0,C 180,E1 -18782.795,E2 -18782.795} C_VEL
LIN {X 0,Y 408.444,Z 350.796,A -85,B 0,C 180,E1 -18784.14,E2 -18784.14} C_VEL
LIN {X 0,Y 414.456,Z 382.401,A -85,B 0,C 180,E1 -18785.247,E2 -18785.247} C_VEL
LIN {X 0,Y 418.09,Z 406.855,A -85,B 0,C 180,E1 -18785.986,E2 -18785.986} C_VEL
LIN {X 0,Y 415.924,Z 489.664,A -85,B 0,C 180,E1 -18787.443,E2 -18787.443} C_VEL
LIN {X 0,Y 414.989,Z 504.097,A -85,B 0,C 180,E1 -18787.879,E2 -18787.879} C_VEL
LIN {X 0,Y 413.456,Z 518.547,A -85,B 0,C 180,E1 -18788.512,E2 -18788.512} C_VEL
LIN {X 0,Y 411.825,Z 532.003,A -85,B 0,C 180,E1 -18789.32,E2 -18789.32} C_VEL
LIN {X 0,Y 410.03,Z 544.544,A -85,B 0,C 180,E1 -18790.285,E2 -18790.285} C_VEL
LIN {X 0,Y 408.016,Z 557,A -85,B 0,C 180,E1 -18791.486,E2 -18791.486} C_VEL
LIN {X 0,Y 406.143,Z 567.226,A -85,B 0,C 180,E1 -18792.695,E2 -18792.695} C_VEL
LIN {X 0,Y 404.292,Z 577.44,A -85,B 0,C 180,E1 -18794.168,E2 -18794.168} C_VEL
LIN {X 0,Y 402.777,Z 585.929,A -85,B 0,C 180,E1 -18795.655,E2 -18795.655} C_VEL
LIN {X 0,Y 401.427,Z 594.087,A -85,B 0,C 180,E1 -18797.405,E2 -18797.405} C_VEL
LIN {X 0,Y 400.499,Z 599.849,A -85,B 0,C 180,E1 -18798.911,E2 -18798.911} C_VEL
LIN {X 0,Y 399.786,Z 604.581,A -85,B 0,C 180,E1 -18800.421,E2 -18800.421} C_VEL
LIN {X 0,Y 399.16,Z 609.53,A -85,B 0,C 180,E1 -18802.44,E2 -18802.44} C_VEL
LIN {X 0,Y 399.072,Z 613.651,A -85,B 0,C 180,E1 -18804.715,E2 -18804.715} C_VEL
LIN {X 0,Y 399.01,Z 618.16,A -85,B 0,C 180,E1 -18806.48,E2 -18806.48} C_VEL
LIN {X 0,Y 399,Z 621.018,A -85,B 0,C 180,E1 -18807.99,E2 -18807.99} C_VEL
LIN {X 0,Y 399.055,Z 622.417,A -85,B 0,C 180,E1 -18808.997,E2 -18808.997} C_VEL
LIN {X 0,Y 398.995,Z 624.082,A -85,B 0,C 180,E1 -18811.008,E2 -18811.008} C_VEL
LIN {X 0,Y 398.92,Z 624.288,A -85,B 0,C 180,E1 -18813.022,E2 -18813.022} C_VEL
LIN {X 0,Y 399.04,Z 623.056,A -85,B 0,C 180,E1 -18815.037,E2 -18815.037} C_VEL
LIN {X 0,Y 399.347,Z 620.393,A -85,B 0,C 180,E1 -18817.055,E2 -18817.055} C_VEL
LIN {X 0,Y 399.931,Z 616.203,A -85,B 0,C 180,E1 -18819.072,E2 -18819.072} C_VEL
LIN {X 0,Y 401.161,Z 610.38,A -85,B 0,C 180,E1 -18821.076,E2 -18821.076} C_VEL
LIN {X 0,Y 402.289,Z 603.862,A -85,B 0,C 180,E1 -18822.827,E2 -18822.827} C_VEL
LIN {X 0,Y 403.949,Z 595.754,A -85,B 0,C 180,E1 -18824.564,E2 -18824.564} C_VEL
LIN {X 0,Y 405.708,Z 587.334,A -85,B 0,C 180,E1 -18826.038,E2 -18826.038} C_VEL
LIN {X 0,Y 407.531,Z 577.281,A -85,B 0,C 180,E1 -18827.507,E2 -18827.507} C_VEL
LIN {X 0,Y 409.669,Z 566.162,A -85,B 0,C 180,E1 -18828.83,E2 -18828.83} C_VEL
LIN {X 0,Y 411.732,Z 553.922,A -85,B 0,C 180,E1 -18830.023,E2 -18830.023} C_VEL
LIN {X 0,Y 413.877,Z 540.397,A -85,B 0,C 180,E1 -18831.077,E2 -18831.077} C_VEL
LIN {X 0,Y 415.597,Z 527.573,A -85,B 0,C 180,E1 -18831.876,E2 -18831.876} C_VEL
LIN {X 0,Y 417.371,Z 512.553,A -85,B 0,C 180,E1 -18832.579,E2 -18832.579} C_VEL
LIN {X 0,Y 418.805,Z 496.622,A -85,B 0,C 180,E1 -18833.093,E2 -18833.093} C_VEL
LIN {X 0,Y 424.284,Z 408.126,A -85,B 0,C 180,E1 -18835.358,E2 -18835.358} C_VEL
LIN {X 0,Y 423.007,Z 390.818,A -85,B 0,C 180,E1 -18836.088,E2 -18836.088} C_VEL
LIN {X 0,Y 420.855,Z 372.893,A -85,B 0,C 180,E1 -18836.976,E2 -18836.976} C_VEL
LIN {X 0,Y 418.014,Z 355.284,A -85,B 0,C 180,E1 -18837.983,E2 -18837.983} C_VEL
LIN {X 0,Y 417.639,Z 352.863,A -85,B 0,C 180,E1 -18838.163,E2 -18838.163} C_VEL
LIN {X 0,Y 417.536,Z 348.955,A -85,B 0,C 180,E1 -18838.524,E2 -18838.524} C_VEL
LIN {X 0,Y 416.045,Z 341.575,A -85,B 0,C 180,E1 -18839.439,E2 -18839.439} C_VEL
LIN {X 0,Y 413.963,Z 332.428,A -85,B 0,C 180,E1 -18840.708,E2 -18840.708} C_VEL
LIN {X 0,Y 412.93,Z 328.534,A -85,B 0,C 180,E1 -18841.325,E2 -18841.325} C_VEL
LIN {X 0,Y 408.155,Z 319.856,A -85,B 0,C 180,E1 -18843.312,E2 -18843.312} C_VEL
LIN {X 0,Y 403.99,Z 312.28,A -85,B 0,C 180,E1 -18845.423,E2 -18845.423} C_VEL
LIN {X 0,Y 401.644,Z 308.87,A -85,B 0,C 180,E1 -18846.658,E2 -18846.658} C_VEL
LIN {X 0,Y 401.191,Z 307.07,A -85,B 0,C 180,E1 -18847.184,E2 -18847.184} C_VEL
LIN {X 0,Y 401.174,Z 307.072,A -85,B 0,C 180,E1 -18850.244,E2 -18850.244} C_VEL
LIN {X 0,Y 401.186,Z 307.068,A -85,B 0,C 180,E1 -18852.918,E2 -18852.918} C_VEL
LIN {X 0,Y 401.224,Z 307.063,A -85,B 0,C 180,E1 -18855.708,E2 -18855.708} C_VEL
LIN {X 0,Y 401.193,Z 307.067,A -85,B 0,C 180,E1 -18858.657,E2 -18858.657} C_VEL
LIN {X 0,Y 401.231,Z 307.066,A -85,B 0,C 180,E1 -18862.337,E2 -18862.337} C_VEL
LIN {X 0,Y 401.251,Z 307.059,A -85,B 0,C 180,E1 -18866.04,E2 -18866.04} C_VEL
LIN {X 0,Y 401.249,Z 307.063,A -85,B 0,C 180,E1 -18869.586,E2 -18869.586} C_VEL
LIN {X 0,Y 401.276,Z 307.175,A -85,B 0,C 180,E1 -18871.745,E2 -18871.745} C_VEL
LIN {X 0,Y 402.119,Z 309.634,A -85,B 0,C 180,E1 -18872.671,E2 -18872.671} C_VEL
LIN {X 0,Y 403.398,Z 312.229,A -85,B 0,C 180,E1 -18873.719,E2 -18873.719} C_VEL
LIN {X 0,Y 406.523,Z 319.39,A -85,B 0,C 180,E1 -18876.217,E2 -18876.217} C_VEL
LIN {X 0,Y 409.312,Z 326.725,A -85,B 0,C 180,E1 -18878.425,E2 -18878.425} C_VEL
LIN {X 0,Y 412.118,Z 335.685,A -85,B 0,C 180,E1 -18880.824,E2 -18880.824} C_VEL
LIN {X 0,Y 414.941,Z 347.151,A -85,B 0,C 180,E1 -18883.542,E2 -18883.542} C_VEL
LIN {X 0,Y 420.164,Z 358.405,A -85,B 0,C 180,E1 -18884.683,E2 -18884.683} C_VEL
LIN {X 0,Y 423.482,Z 373.632,A -85,B 0,C 180,E1 -18885.635,E2 -18885.635} C_VEL
LIN {X 0,Y 425.8,Z 388.037,A -85,B 0,C 180,E1 -18886.394,E2 -18886.394} C_VEL
LIN {X 0,Y 419.296,Z 488.526,A -85,B 0,C 180,E1 -18888.954,E2 -18888.954} C_VEL
LIN {X 0,Y 417.866,Z 503.927,A -85,B 0,C 180,E1 -18889.558,E2 -18889.558} C_VEL
LIN {X 0,Y 416.282,Z 517.977,A -85,B 0,C 180,E1 -18890.313,E2 -18890.313} C_VEL
LIN {X 0,Y 414.343,Z 531.619,A -85,B 0,C 180,E1 -18891.249,E2 -18891.249} C_VEL
LIN {X 0,Y 412.154,Z 545.111,A -85,B 0,C 180,E1 -18892.432,E2 -18892.432} C_VEL
LIN {X 0,Y 410.019,Z 557.214,A -85,B 0,C 180,E1 -18893.748,E2 -18893.748} C_VEL
LIN {X 0,Y 408.127,Z 567.221,A -85,B 0,C 180,E1 -18895.077,E2 -18895.077} C_VEL
LIN {X 0,Y 406.275,Z 576.395,A -85,B 0,C 180,E1 -18896.541,E2 -18896.541} C_VEL
LIN {X 0,Y 404.188,Z 585.23,A -85,B 0,C 180,E1 -18898.262,E2 -18898.262} C_VEL
LIN {X 0,Y 402.645,Z 592.326,A -85,B 0,C 180,E1 -18900,E2 -18900} C_VEL
LIN {X 0,Y 401.535,Z 597.294,A -85,B 0,C 180,E1 -18901.499,E2 -18901.499} C_VEL
LIN {X 0,Y 400.653,Z 601.274,A -85,B 0,C 180,E1 -18903.006,E2 -18903.006} C_VEL
LIN {X 0,Y 399.958,Z 605.192,A -85,B 0,C 180,E1 -18905.023,E2 -18905.023} C_VEL
LIN {X 0,Y 399.28,Z 607.624,A -85,B 0,C 180,E1 -18907.054,E2 -18907.054} C_VEL
LIN {X 0,Y 398.951,Z 608.609,A -85,B 0,C 180,E1 -18909.092,E2 -18909.092} C_VEL
LIN {X 0,Y 398.852,Z 608.493,A -85,B 0,C 180,E1 -18910.432,E2 -18910.432} C_VEL
LIN {X 0,Y 398.687,Z 607.356,A -85,B 0,C 180,E1 -18912.171,E2 -18912.171} C_VEL
LIN {X 0,Y 398.768,Z 604.631,A -85,B 0,C 180,E1 -18914.236,E2 -18914.236} C_VEL
LIN {X 0,Y 398.888,Z 601.484,A -85,B 0,C 180,E1 -18915.794,E2 -18915.794} C_VEL
LIN {X 0,Y 399.063,Z 597.34,A -85,B 0,C 180,E1 -18917.361,E2 -18917.361} C_VEL
LIN {X 0,Y 399.319,Z 592.031,A -85,B 0,C 180,E1 -18918.954,E2 -18918.954} C_VEL
LIN {X 0,Y 399.75,Z 584.408,A -85,B 0,C 180,E1 -18920.783,E2 -18920.783} C_VEL
LIN {X 0,Y 400.263,Z 575.969,A -85,B 0,C 180,E1 -18922.419,E2 -18922.419} C_VEL
LIN {X 0,Y 400.942,Z 566.247,A -85,B 0,C 180,E1 -18923.965,E2 -18923.965} C_VEL
LIN {X 0,Y 401.715,Z 555.043,A -85,B 0,C 180,E1 -18925.427,E2 -18925.427} C_VEL
LIN {X 0,Y 402.632,Z 542.65,A -85,B 0,C 180,E1 -18926.753,E2 -18926.753} C_VEL
LIN {X 0,Y 403.466,Z 530.102,A -85,B 0,C 180,E1 -18927.846,E2 -18927.846} C_VEL
LIN {X 0,Y 404.272,Z 516.192,A -85,B 0,C 180,E1 -18928.808,E2 -18928.808} C_VEL
LIN {X 0,Y 405.101,Z 501.366,A -85,B 0,C 180,E1 -18929.595,E2 -18929.595} C_VEL
LIN {X 0,Y 405.845,Z 486.337,A -85,B 0,C 180,E1 -18930.168,E2 -18930.168} C_VEL
LIN {X 0,Y 406.684,Z 450.363,A -85,B 0,C 180,E1 -18931.028,E2 -18931.028} C_VEL
LIN {X 0,Y 408.674,Z 377.652,A -85,B 0,C 180,E1 -18932.705,E2 -18932.705} C_VEL
LIN {X 0,Y 404.64,Z 344.795,A -85,B 0,C 180,E1 -18933.637,E2 -18933.637} C_VEL
LIN {X 0,Y 405.527,Z 330.167,A -85,B 0,C 180,E1 -18935.963,E2 -18935.963} C_VEL
LIN {X 0,Y 405.107,Z 326.209,A -85,B 0,C 180,E1 -18936.621,E2 -18936.621} C_VEL
LIN {X 0,Y 401.26,Z 307.06,A -85,B 0,C 180,E1 -18939.941,E2 -18939.941} C_VEL
LIN {X 0,Y 401.204,Z 307.065,A -85,B 0,C 180,E1 -18942.913,E2 -18942.913} C_VEL
LIN {X 0,Y 401.223,Z 307.06,A -85,B 0,C 180,E1 -18945.706,E2 -18945.706} C_VEL
LIN {X 0,Y 401.187,Z 307.068,A -85,B 0,C 180,E1 -18948.655,E2 -18948.655} C_VEL
LIN {X 0,Y 401.214,Z 307.068,A -85,B 0,C 180,E1 -18952.333,E2 -18952.333} C_VEL
LIN {X 0,Y 401.214,Z 307.064,A -85,B 0,C 180,E1 -18956.035,E2 -18956.035} C_VEL
LIN {X 0,Y 401.221,Z 307.063,A -85,B 0,C 180,E1 -18959.582,E2 -18959.582} C_VEL
LIN {X 0,Y 401.248,Z 307.057,A -85,B 0,C 180,E1 -18963.005,E2 -18963.005} C_VEL
LIN {X 0,Y 401.265,Z 307.06,A -85,B 0,C 180,E1 -18966.327,E2 -18966.327} C_VEL
LIN {X 0,Y 401.277,Z 307.057,A -85,B 0,C 180,E1 -18969.565,E2 -18969.565} C_VEL
LIN {X 0,Y 401.31,Z 307.05,A -85,B 0,C 180,E1 -18972.737,E2 -18972.737} C_VEL
LIN {X 0,Y 401.349,Z 307.052,A -85,B 0,C 180,E1 -18975.855,E2 -18975.855} C_VEL
LIN {X 0,Y 401.429,Z 307.037,A -85,B 0,C 180,E1 -18978.932,E2 -18978.932} C_VEL
LIN {X 0,Y 401.413,Z 307.042,A -85,B 0,C 180,E1 -18979.071,E2 -18979.071} C_VEL
LIN {X 0,Y 401.82,Z 309.243,A -85,B 0,C 180,E1 -18979.623,E2 -18979.623} C_VEL
LIN {X 0,Y 409.932,Z 333.809,A -85,B 0,C 180,E1 -18980.461,E2 -18980.461} C_VEL
LIN {X 0,Y 410.776,Z 337.885,A -85,B 0,C 180,E1 -18980.574,E2 -18980.574} C_VEL
LIN {X 0,Y 408.632,Z 445.383,A -85,B 0,C 180,E1 -18982.457,E2 -18982.457} C_VEL
LIN {X 0,Y 408.162,Z 459.662,A -85,B 0,C 180,E1 -18982.913,E2 -18982.913} C_VEL
LIN {X 0,Y 407.472,Z 473.969,A -85,B 0,C 180,E1 -18983.582,E2 -18983.582} C_VEL
LIN {X 0,Y 406.564,Z 487.568,A -85,B 0,C 180,E1 -18984.436,E2 -18984.436} C_VEL
LIN {X 0,Y 405.703,Z 498.385,A -85,B 0,C 180,E1 -18985.294,E2 -18985.294} C_VEL
LIN {X 0,Y 404.48,Z 509.896,A -85,B 0,C 180,E1 -18986.399,E2 -18986.399} C_VEL
LIN {X 0,Y 403.714,Z 519.407,A -85,B 0,C 180,E1 -18987.512,E2 -18987.512} C_VEL
LIN {X 0,Y 402.793,Z 528.4,A -85,B 0,C 180,E1 -18988.752,E2 -18988.752} C_VEL
LIN {X 0,Y 401.77,Z 537.451,A -85,B 0,C 180,E1 -18990.247,E2 -18990.247} C_VEL
LIN {X 0,Y 401.006,Z 544.984,A -85,B 0,C 180,E1 -18991.749,E2 -18991.749} C_VEL
LIN {X 0,Y 400.532,Z 550.278,A -85,B 0,C 180,E1 -18993.005,E2 -18993.005} C_VEL
LIN {X 0,Y 400.227,Z 555.61,A -85,B 0,C 180,E1 -18994.514,E2 -18994.514} C_VEL
LIN {X 0,Y 399.674,Z 561.274,A -85,B 0,C 180,E1 -18996.538,E2 -18996.538} C_VEL
LIN {X 0,Y 399.344,Z 564.487,A -85,B 0,C 180,E1 -18998.064,E2 -18998.064} C_VEL
LIN {X 0,Y 399.258,Z 567.488,A -85,B 0,C 180,E1 -19000.101,E2 -19000.101} C_VEL
LIN {X 0,Y 399.189,Z 569.131,A -85,B 0,C 180,E1 -19002.152,E2 -19002.152} C_VEL
LIN {X 0,Y 399.401,Z 569.417,A -85,B 0,C 180,E1 -19004.21,E2 -19004.21} C_VEL
LIN {X 0,Y 399.741,Z 568.349,A -85,B 0,C 180,E1 -19006.279,E2 -19006.279} C_VEL
LIN {X 0,Y 400.312,Z 565.884,A -85,B 0,C 180,E1 -19008.355,E2 -19008.355} C_VEL
LIN {X 0,Y 401.203,Z 561.888,A -85,B 0,C 180,E1 -19010.434,E2 -19010.434} C_VEL
LIN {X 0,Y 402.378,Z 556.246,A -85,B 0,C 180,E1 -19012.515,E2 -19012.515} C_VEL
LIN {X 0,Y 403.724,Z 549.805,A -85,B 0,C 180,E1 -19014.331,E2 -19014.331} C_VEL
LIN {X 0,Y 405.333,Z 542.248,A -85,B 0,C 180,E1 -19016.026,E2 -19016.026} C_VEL
LIN {X 0,Y 407.051,Z 533.167,A -85,B 0,C 180,E1 -19017.682,E2 -19017.682} C_VEL
LIN {X 0,Y 408.798,Z 523.676,A -85,B 0,C 180,E1 -19019.091,E2 -19019.091} C_VEL
LIN {X 0,Y 410.5,Z 513.333,A -85,B 0,C 180,E1 -19020.361,E2 -19020.361} C_VEL
LIN {X 0,Y 412.169,Z 502.017,A -85,B 0,C 180,E1 -19021.501,E2 -19021.501} C_VEL
LIN {X 0,Y 413.739,Z 489.66,A -85,B 0,C 180,E1 -19022.506,E2 -19022.506} C_VEL
LIN {X 0,Y 413.896,Z 488.141,A -85,B 0,C 180,E1 -19022.611,E2 -19022.611} C_VEL
LIN {X 0,Y 413.867,Z 482.93,A -85,B 0,C 180,E1 -19023.003,E2 -19023.003} C_VEL
LIN {X 0,Y 411.958,Z 474.494,A -85,B 0,C 180,E1 -19023.686,E2 -19023.686} C_VEL
LIN {X 0,Y 410.099,Z 465.837,A -85,B 0,C 180,E1 -19024.299,E2 -19024.299} C_VEL
LIN {X 0,Y 409.957,Z 460.294,A -85,B 0,C 180,E1 -19024.563,E2 -19024.563} C_VEL
LIN {X 0,Y 410.622,Z 446.973,A -85,B 0,C 180,E1 -19024.988,E2 -19024.988} C_VEL
LIN {X 0,Y 411.708,Z 405.019,A -85,B 0,C 180,E1 -19025.763,E2 -19025.763} C_VEL
LIN {X 0,Y 413.183,Z 350.058,A -85,B 0,C 180,E1 -19026.727,E2 -19026.727} C_VEL
LIN {X 0,Y 404.61,Z 330.67,A -85,B 0,C 180,E1 -19027.804,E2 -19027.804} C_VEL
LIN {X 0,Y 396.219,Z 314.088,A -85,B 0,C 180,E1 -19028.866,E2 -19028.866} C_VEL
LIN {X 0,Y 394.914,Z 311.265,A -85,B 0,C 180,E1 -19029.069,E2 -19029.069} C_VEL
LIN {X 0,Y 394.129,Z 307.953,A -85,B 0,C 180,E1 -19030.077,E2 -19030.077} C_VEL
LIN {X 0,Y 394.127,Z 307.952,A -85,B 0,C 180,E1 -19033.226,E2 -19033.226} C_VEL
LIN {X 0,Y 394.158,Z 307.938,A -85,B 0,C 180,E1 -19036.128,E2 -19036.128} C_VEL
LIN {X 0,Y 394.132,Z 307.946,A -85,B 0,C 180,E1 -19039.83,E2 -19039.83} C_VEL
LIN {X 0,Y 394.164,Z 307.926,A -85,B 0,C 180,E1 -19043.093,E2 -19043.093} C_VEL
LIN {X 0,Y 394.176,Z 307.919,A -85,B 0,C 180,E1 -19045.345,E2 -19045.345} C_VEL
LIN {X 0,Y 394.169,Z 307.935,A -85,B 0,C 180,E1 -19048.98,E2 -19048.98} C_VEL
LIN {X 0,Y 394.18,Z 307.944,A -85,B 0,C 180,E1 -19051.329,E2 -19051.329} C_VEL
LIN {X 0,Y 394.198,Z 307.939,A -85,B 0,C 180,E1 -19054.757,E2 -19054.757} C_VEL
LIN {X 0,Y 394.212,Z 307.938,A -85,B 0,C 180,E1 -19058.091,E2 -19058.091} C_VEL
LIN {X 0,Y 394.22,Z 307.925,A -85,B 0,C 180,E1 -19061.348,E2 -19061.348} C_VEL
LIN {X 0,Y 394.25,Z 307.93,A -85,B 0,C 180,E1 -19064.544,E2 -19064.544} C_VEL
LIN {X 0,Y 394.39,Z 307.916,A -85,B 0,C 180,E1 -19067.695,E2 -19067.695} C_VEL
LIN {X 0,Y 394.406,Z 307.903,A -85,B 0,C 180,E1 -19071.832,E2 -19071.832} C_VEL
LIN {X 0,Y 394.508,Z 307.896,A -85,B 0,C 180,E1 -19074.907,E2 -19074.907} C_VEL
LIN {X 0,Y 394.422,Z 307.908,A -85,B 0,C 180,E1 -19077.965,E2 -19077.965} C_VEL
LIN {X 0,Y 394.424,Z 307.898,A -85,B 0,C 180,E1 -19081.018,E2 -19081.018} C_VEL
LIN {X 0,Y 394.529,Z 307.895,A -85,B 0,C 180,E1 -19084.072,E2 -19084.072} C_VEL
LIN {X 0,Y 394.429,Z 307.894,A -85,B 0,C 180,E1 -19087.141,E2 -19087.141} C_VEL
LIN {X 0,Y 394.362,Z 307.915,A -85,B 0,C 180,E1 -19090.231,E2 -19090.231} C_VEL
LIN {X 0,Y 394.394,Z 307.898,A -85,B 0,C 180,E1 -19092.381,E2 -19092.381} C_VEL
LIN {X 0,Y 394.284,Z 307.918,A -85,B 0,C 180,E1 -19096.513,E2 -19096.513} C_VEL
LIN {X 0,Y 394.249,Z 307.929,A -85,B 0,C 180,E1 -19099.729,E2 -19099.729} C_VEL
LIN {X 0,Y 394.188,Z 307.932,A -85,B 0,C 180,E1 -19103.012,E2 -19103.012} C_VEL
LIN {X 0,Y 394.201,Z 307.93,A -85,B 0,C 180,E1 -19106.373,E2 -19106.373} C_VEL
LIN {X 0,Y 394.205,Z 307.934,A -85,B 0,C 180,E1 -19109.836,E2 -19109.836} C_VEL
LIN {X 0,Y 394.179,Z 307.937,A -85,B 0,C 180,E1 -19113.426,E2 -19113.426} C_VEL
LIN {X 0,Y 394.246,Z 307.908,A -85,B 0,C 180,E1 -19116.923,E2 -19116.923} C_VEL
LIN {X 0,Y 394.184,Z 307.937,A -85,B 0,C 180,E1 -19120.179,E2 -19120.179} C_VEL
LIN {X 0,Y 394.205,Z 307.939,A -85,B 0,C 180,E1 -19123.866,E2 -19123.866} C_VEL
LIN {X 0,Y 394.166,Z 307.942,A -85,B 0,C 180,E1 -19126.768,E2 -19126.768} C_VEL
LIN {X 0,Y 394.203,Z 307.943,A -85,B 0,C 180,E1 -19130.237,E2 -19130.237} C_VEL
LIN {X 0,Y 394.278,Z 308.022,A -85,B 0,C 180,E1 -19133.679,E2 -19133.679} C_VEL
LIN {X 0,Y 397.515,Z 320.585,A -85,B 0,C 180,E1 -19136.894,E2 -19136.894} C_VEL
LIN {X 0,Y 400.626,Z 334.139,A -85,B 0,C 180,E1 -19140.117,E2 -19140.117} C_VEL
LIN {X 0,Y 402.672,Z 344.846,A -85,B 0,C 180,E1 -19142.516,E2 -19142.516} C_VEL
LIN {X 0,Y 401.908,Z 350.472,A -85,B 0,C 180,E1 -19143.618,E2 -19143.618} C_VEL
LIN {X 0,Y 408.249,Z 383.712,A -85,B 0,C 180,E1 -19144.801,E2 -19144.801} C_VEL
LIN {X 0,Y 411.821,Z 407.926,A -85,B 0,C 180,E1 -19145.548,E2 -19145.548} C_VEL
LIN {X 0,Y 409.557,Z 489.599,A -85,B 0,C 180,E1 -19147.006,E2 -19147.006} C_VEL
LIN {X 0,Y 408.591,Z 503.915,A -85,B 0,C 180,E1 -19147.448,E2 -19147.448} C_VEL
LIN {X 0,Y 407.028,Z 518.302,A -85,B 0,C 180,E1 -19148.089,E2 -19148.089} C_VEL
LIN {X 0,Y 405.349,Z 531.767,A -85,B 0,C 180,E1 -19148.911,E2 -19148.911} C_VEL
LIN {X 0,Y 403.588,Z 543.528,A -85,B 0,C 180,E1 -19149.825,E2 -19149.825} C_VEL
LIN {X 0,Y 401.699,Z 554.923,A -85,B 0,C 180,E1 -19150.919,E2 -19150.919} C_VEL
LIN {X 0,Y 399.742,Z 565.423,A -85,B 0,C 180,E1 -19152.146,E2 -19152.146} C_VEL
LIN {X 0,Y 397.728,Z 575.886,A -85,B 0,C 180,E1 -19153.636,E2 -19153.636} C_VEL
LIN {X 0,Y 395.885,Z 585.871,A -85,B 0,C 180,E1 -19155.399,E2 -19155.399} C_VEL
LIN {X 0,Y 394.467,Z 593.954,A -85,B 0,C 180,E1 -19157.179,E2 -19157.179} C_VEL
LIN {X 0,Y 393.501,Z 599.681,A -85,B 0,C 180,E1 -19158.711,E2 -19158.711} C_VEL
LIN {X 0,Y 392.564,Z 605.738,A -85,B 0,C 180,E1 -19160.762,E2 -19160.762} C_VEL
LIN {X 0,Y 392.032,Z 610.239,A -85,B 0,C 180,E1 -19162.818,E2 -19162.818} C_VEL
LIN {X 0,Y 391.981,Z 613.367,A -85,B 0,C 180,E1 -19164.748,E2 -19164.748} C_VEL
LIN {X 0,Y 391.932,Z 617.629,A -85,B 0,C 180,E1 -19166.416,E2 -19166.416} C_VEL
LIN {X 0,Y 391.926,Z 620.598,A -85,B 0,C 180,E1 -19167.954,E2 -19167.954} C_VEL
LIN {X 0,Y 391.979,Z 622.059,A -85,B 0,C 180,E1 -19168.979,E2 -19168.979} C_VEL
LIN {X 0,Y 391.908,Z 623.84,A -85,B 0,C 180,E1 -19171.027,E2 -19171.027} C_VEL
LIN {X 0,Y 391.82,Z 624.159,A -85,B 0,C 180,E1 -19173.077,E2 -19173.077} C_VEL
LIN {X 0,Y 391.949,Z 623.044,A -85,B 0,C 180,E1 -19175.129,E2 -19175.129} C_VEL
LIN {X 0,Y 392.285,Z 620.495,A -85,B 0,C 180,E1 -19177.182,E2 -19177.182} C_VEL
LIN {X 0,Y 392.931,Z 616.48,A -85,B 0,C 180,E1 -19179.235,E2 -19179.235} C_VEL
LIN {X 0,Y 393.837,Z 612.375,A -85,B 0,C 180,E1 -19180.765,E2 -19180.765} C_VEL
LIN {X 0,Y 394.969,Z 606.401,A -85,B 0,C 180,E1 -19182.552,E2 -19182.552} C_VEL
LIN {X 0,Y 396.614,Z 598.973,A -85,B 0,C 180,E1 -19184.317,E2 -19184.317} C_VEL
LIN {X 0,Y 398.302,Z 591.206,A -85,B 0,C 180,E1 -19185.82,E2 -19185.82} C_VEL
LIN {X 0,Y 400.204,Z 581.981,A -85,B 0,C 180,E1 -19187.312,E2 -19187.312} C_VEL
LIN {X 0,Y 402.222,Z 571.866,A -85,B 0,C 180,E1 -19188.664,E2 -19188.664} C_VEL
LIN {X 0,Y 404.539,Z 559.645,A -85,B 0,C 180,E1 -19189.999,E2 -19189.999} C_VEL
LIN {X 0,Y 406.679,Z 547.505,A -85,B 0,C 180,E1 -19191.074,E2 -19191.074} C_VEL
LIN {X 0,Y 408.706,Z 534.253,A -85,B 0,C 180,E1 -19192.02,E2 -19192.02} C_VEL
LIN {X 0,Y 410.638,Z 520.198,A -85,B 0,C 180,E1 -19192.799,E2 -19192.799} C_VEL
LIN {X 0,Y 412.294,Z 505.268,A -85,B 0,C 180,E1 -19193.401,E2 -19193.401} C_VEL
LIN {X 0,Y 413.74,Z 484.674,A -85,B 0,C 180,E1 -19193.975,E2 -19193.975} C_VEL
LIN {X 0,Y 418.752,Z 409.424,A -85,B 0,C 180,E1 -19195.941,E2 -19195.941} C_VEL
LIN {X 0,Y 417.626,Z 392.724,A -85,B 0,C 180,E1 -19196.665,E2 -19196.665} C_VEL
LIN {X 0,Y 415.746,Z 375.864,A -85,B 0,C 180,E1 -19197.518,E2 -19197.518} C_VEL
LIN {X 0,Y 412.977,Z 357.892,A -85,B 0,C 180,E1 -19198.577,E2 -19198.577} C_VEL
LIN {X 0,Y 412.183,Z 353.094,A -85,B 0,C 180,E1 -19198.903,E2 -19198.903} C_VEL
LIN {X 0,Y 411.521,Z 348.205,A -85,B 0,C 180,E1 -19199.47,E2 -19199.47} C_VEL
LIN {X 0,Y 408.981,Z 336.647,A -85,B 0,C 180,E1 -19201.093,E2 -19201.093} C_VEL
LIN {X 0,Y 407.752,Z 332.67,A -85,B 0,C 180,E1 -19201.765,E2 -19201.765} C_VEL
LIN {X 0,Y 403.57,Z 324.985,A -85,B 0,C 180,E1 -19203.581,E2 -19203.581} C_VEL
LIN {X 0,Y 399.363,Z 317.384,A -85,B 0,C 180,E1 -19205.762,E2 -19205.762} C_VEL
LIN {X 0,Y 397.418,Z 314.454,A -85,B 0,C 180,E1 -19206.818,E2 -19206.818} C_VEL
LIN {X 0,Y 396.756,Z 312.594,A -85,B 0,C 180,E1 -19207.397,E2 -19207.397} C_VEL
LIN {X 0,Y 394.759,Z 310.036,A -85,B 0,C 180,E1 -19208.674,E2 -19208.674} C_VEL
LIN {X 0,Y 394.128,Z 307.948,A -85,B 0,C 180,E1 -19209.411,E2 -19209.411} C_VEL
LIN {X 0,Y 394.121,Z 307.946,A -85,B 0,C 180,E1 -19212.484,E2 -19212.484} C_VEL
LIN {X 0,Y 394.162,Z 307.941,A -85,B 0,C 180,E1 -19215.304,E2 -19215.304} C_VEL
LIN {X 0,Y 394.138,Z 307.947,A -85,B 0,C 180,E1 -19218.887,E2 -19218.887} C_VEL
LIN {X 0,Y 394.183,Z 307.941,A -85,B 0,C 180,E1 -19221.542,E2 -19221.542} C_VEL
LIN {X 0,Y 394.219,Z 307.937,A -85,B 0,C 180,E1 -19224.821,E2 -19224.821} C_VEL
LIN {X 0,Y 394.188,Z 307.94,A -85,B 0,C 180,E1 -19228.535,E2 -19228.535} C_VEL
LIN {X 0,Y 394.222,Z 308.063,A -85,B 0,C 180,E1 -19229.651,E2 -19229.651} C_VEL
LIN {X 0,Y 395.257,Z 310.779,A -85,B 0,C 180,E1 -19230.906,E2 -19230.906} C_VEL
LIN {X 0,Y 396.029,Z 311.818,A -85,B 0,C 180,E1 -19231.475,E2 -19231.475} C_VEL
LIN {X 0,Y 399.363,Z 319.605,A -85,B 0,C 180,E1 -19234.588,E2 -19234.588} C_VEL
LIN {X 0,Y 402.513,Z 327.65,A -85,B 0,C 180,E1 -19237.268,E2 -19237.268} C_VEL
LIN {X 0,Y 405.408,Z 336.357,A -85,B 0,C 180,E1 -19239.785,E2 -19239.785} C_VEL
LIN {X 0,Y 407.689,Z 345.004,A -85,B 0,C 180,E1 -19241.986,E2 -19241.986} C_VEL
LIN {X 0,Y 408.425,Z 347.884,A -85,B 0,C 180,E1 -19242.629,E2 -19242.629} C_VEL
LIN {X 0,Y 412.769,Z 356.365,A -85,B 0,C 180,E1 -19243.608,E2 -19243.608} C_VEL
LIN {X 0,Y 415.495,Z 362.806,A -85,B 0,C 180,E1 -19244.231,E2 -19244.231} C_VEL
LIN {X 0,Y 418.326,Z 376.736,A -85,B 0,C 180,E1 -19245.114,E2 -19245.114} C_VEL
LIN {X 0,Y 420.303,Z 389.657,A -85,B 0,C 180,E1 -19245.811,E2 -19245.811} C_VEL
LIN {X 0,Y 413.504,Z 488.95,A -85,B 0,C 180,E1 -19248.396,E2 -19248.396} C_VEL
LIN {X 0,Y 412.08,Z 503.591,A -85,B 0,C 180,E1 -19248.976,E2 -19248.976} C_VEL
LIN {X 0,Y 410.279,Z 518.647,A -85,B 0,C 180,E1 -19249.798,E2 -19249.798} C_VEL
LIN {X 0,Y 408.248,Z 532.138,A -85,B 0,C 180,E1 -19250.744,E2 -19250.744} C_VEL
LIN {X 0,Y 406.19,Z 544.346,A -85,B 0,C 180,E1 -19251.821,E2 -19251.821} C_VEL
LIN {X 0,Y 403.893,Z 556.576,A -85,B 0,C 180,E1 -19253.152,E2 -19253.152} C_VEL
LIN {X 0,Y 401.943,Z 566.45,A -85,B 0,C 180,E1 -19254.463,E2 -19254.463} C_VEL
LIN {X 0,Y 399.929,Z 575.965,A -85,B 0,C 180,E1 -19255.983,E2 -19255.983} C_VEL
